LIN {X 0,Y 736.1,Z 322.543,A -85,B 0,C 180,E1 33323.915,E2 33323.915} C_VEL
LIN {X 0,Y 736.031,Z 322.542,A -85,B 0,C 180,E1 33321.184,E2 33321.184} C_VEL
LIN {X 0,Y 736.024,Z 322.538,A -85,B 0,C 180,E1 33318.7,E2 33318.7} C_VEL
LIN {X 0,Y 736.098,Z 322.534,A -85,B 0,C 180,E1 33315.911,E2 33315.911} C_VEL
LIN {X 0,Y 736.039,Z 322.537,A -85,B 0,C 180,E1 33313.033,E2 33313.033} C_VEL
LIN {X 0,Y 736.026,Z 322.539,A -85,B 0,C 180,E1 33310.489,E2 33310.489} C_VEL
LIN {X 0,Y 736.094,Z 322.535,A -85,B 0,C 180,E1 33307.729,E2 33307.729} C_VEL
LIN {X 0,Y 736.045,Z 322.543,A -85,B 0,C 180,E1 33304.831,E2 33304.831} C_VEL
LIN {X 0,Y 736.027,Z 322.536,A -85,B 0,C 180,E1 33302.258,E2 33302.258} C_VEL
LIN {X 0,Y 736.094,Z 322.533,A -85,B 0,C 180,E1 33299.533,E2 33299.533} C_VEL
LIN {X 0,Y 736.044,Z 322.536,A -85,B 0,C 180,E1 33296.573,E2 33296.573} C_VEL
LIN {X 0,Y 736.031,Z 322.539,A -85,B 0,C 180,E1 33293.996,E2 33293.996} C_VEL
LIN {X 0,Y 736.097,Z 322.534,A -85,B 0,C 180,E1 33291.249,E2 33291.249} C_VEL
LIN {X 0,Y 736.097,Z 322.534,A -85,B 0,C 180,E1 33289.048,E2 33289.048} C_VEL
LIN {X 0,Y 735.115,Z 322.666,A -85,B 0,C 180,E1 33288.448,E2 33288.448} C_VEL
LIN {X 0,Y 728.677,Z 323.466,A -85,B 0,C 180,E1 33286.769,E2 33286.769} C_VEL
LIN {X 0,Y 728.112,Z 323.525,A -85,B 0,C 180,E1 33286.333,E2 33286.333} C_VEL
LIN {X 0,Y 728.094,Z 323.528,A -85,B 0,C 180,E1 33283.72,E2 33283.72} C_VEL
LIN {X 0,Y 728.157,Z 323.522,A -85,B 0,C 180,E1 33280.924,E2 33280.924} C_VEL
LIN {X 0,Y 728.106,Z 323.53,A -85,B 0,C 180,E1 33277.981,E2 33277.981} C_VEL
LIN {X 0,Y 728.098,Z 323.526,A -85,B 0,C 180,E1 33275.379,E2 33275.379} C_VEL
LIN {X 0,Y 728.159,Z 323.527,A -85,B 0,C 180,E1 33272.504,E2 33272.504} C_VEL
LIN {X 0,Y 728.102,Z 323.53,A -85,B 0,C 180,E1 33269.644,E2 33269.644} C_VEL
LIN {X 0,Y 728.107,Z 323.529,A -85,B 0,C 180,E1 33267.039,E2 33267.039} C_VEL
LIN {X 0,Y 728.16,Z 323.531,A -85,B 0,C 180,E1 33264.102,E2 33264.102} C_VEL
LIN {X 0,Y 728.107,Z 323.58,A -85,B 0,C 180,E1 33261.311,E2 33261.311} C_VEL
LIN {X 0,Y 729.232,Z 326.748,A -85,B 0,C 180,E1 33260.997,E2 33260.997} C_VEL
LIN {X 0,Y 733.452,Z 336.26,A -85,B 0,C 180,E1 33260.007,E2 33260.007} C_VEL
LIN {X 0,Y 733.535,Z 341.384,A -85,B 0,C 180,E1 33259.674,E2 33259.674} C_VEL
LIN {X 0,Y 735.852,Z 350.383,A -85,B 0,C 180,E1 33259.391,E2 33259.391} C_VEL
LIN {X 0,Y 734.942,Z 560.635,A -85,B 0,C 180,E1 33256.782,E2 33256.782} C_VEL
LIN {X 0,Y 734.06,Z 784.489,A -85,B 0,C 180,E1 33254.097,E2 33254.097} C_VEL
LIN {X 0,Y 733.842,Z 824.081,A -85,B 0,C 180,E1 33253.594,E2 33253.594} C_VEL
LIN {X 0,Y 733.512,Z 850.633,A -85,B 0,C 180,E1 33253.099,E2 33253.099} C_VEL
LIN {X 0,Y 733.193,Z 876.497,A -85,B 0,C 180,E1 33252.467,E2 33252.467} C_VEL
LIN {X 0,Y 732.75,Z 904.112,A -85,B 0,C 180,E1 33251.617,E2 33251.617} C_VEL
LIN {X 0,Y 732.239,Z 928.977,A -85,B 0,C 180,E1 33250.694,E2 33250.694} C_VEL
LIN {X 0,Y 731.795,Z 951.691,A -85,B 0,C 180,E1 33249.712,E2 33249.712} C_VEL
LIN {X 0,Y 731.337,Z 975.92,A -85,B 0,C 180,E1 33248.517,E2 33248.517} C_VEL
LIN {X 0,Y 730.768,Z 999.778,A -85,B 0,C 180,E1 33247.162,E2 33247.162} C_VEL
LIN {X 0,Y 730.337,Z 1020.658,A -85,B 0,C 180,E1 33245.826,E2 33245.826} C_VEL
LIN {X 0,Y 729.892,Z 1043.125,A -85,B 0,C 180,E1 33244.217,E2 33244.217} C_VEL
LIN {X 0,Y 729.439,Z 1063.156,A -85,B 0,C 180,E1 33242.595,E2 33242.595} C_VEL
LIN {X 0,Y 729.121,Z 1082.465,A -85,B 0,C 180,E1 33240.854,E2 33240.854} C_VEL
LIN {X 0,Y 728.788,Z 1100.104,A -85,B 0,C 180,E1 33239.056,E2 33239.056} C_VEL
LIN {X 0,Y 728.566,Z 1114.981,A -85,B 0,C 180,E1 33237.37,E2 33237.37} C_VEL
LIN {X 0,Y 728.345,Z 1130.773,A -85,B 0,C 180,E1 33235.36,E2 33235.36} C_VEL
LIN {X 0,Y 728.172,Z 1143.719,A -85,B 0,C 180,E1 33233.466,E2 33233.466} C_VEL
LIN {X 0,Y 728.099,Z 1154.015,A -85,B 0,C 180,E1 33231.763,E2 33231.763} C_VEL
LIN {X 0,Y 728.021,Z 1163.405,A -85,B 0,C 180,E1 33229.997,E2 33229.997} C_VEL
LIN {X 0,Y 727.956,Z 1173.511,A -85,B 0,C 180,E1 33227.753,E2 33227.753} C_VEL
LIN {X 0,Y 727.938,Z 1181.236,A -85,B 0,C 180,E1 33225.618,E2 33225.618} C_VEL
LIN {X 0,Y 727.921,Z 1187.251,A -85,B 0,C 180,E1 33223.46,E2 33223.46} C_VEL
LIN {X 0,Y 727.912,Z 1191.364,A -85,B 0,C 180,E1 33221.408,E2 33221.408} C_VEL
LIN {X 0,Y 727.912,Z 1193.964,A -85,B 0,C 180,E1 33219.328,E2 33219.328} C_VEL
LIN {X 0,Y 727.912,Z 1194.92,A -85,B 0,C 180,E1 33217.26,E2 33217.26} C_VEL
LIN {X 0,Y 727.914,Z 1194.252,A -85,B 0,C 180,E1 33214.964,E2 33214.964} C_VEL
LIN {X 0,Y 727.911,Z 1192.016,A -85,B 0,C 180,E1 33212.913,E2 33212.913} C_VEL
LIN {X 0,Y 727.916,Z 1187.872,A -85,B 0,C 180,E1 33210.708,E2 33210.708} C_VEL
LIN {X 0,Y 727.926,Z 1182.373,A -85,B 0,C 180,E1 33208.662,E2 33208.662} C_VEL
LIN {X 0,Y 727.944,Z 1175.333,A -85,B 0,C 180,E1 33206.614,E2 33206.614} C_VEL
LIN {X 0,Y 728.001,Z 1165.854,A -85,B 0,C 180,E1 33204.404,E2 33204.404} C_VEL
LIN {X 0,Y 728.074,Z 1155.152,A -85,B 0,C 180,E1 33202.345,E2 33202.345} C_VEL
LIN {X 0,Y 728.186,Z 1144.682,A -85,B 0,C 180,E1 33200.596,E2 33200.596} C_VEL
LIN {X 0,Y 728.307,Z 1133.374,A -85,B 0,C 180,E1 33198.919,E2 33198.919} C_VEL
LIN {X 0,Y 728.51,Z 1118.777,A -85,B 0,C 180,E1 33196.992,E2 33196.992} C_VEL
LIN {X 0,Y 728.753,Z 1102.69,A -85,B 0,C 180,E1 33195.134,E2 33195.134} C_VEL
LIN {X 0,Y 729.006,Z 1086.805,A -85,B 0,C 180,E1 33193.484,E2 33193.484} C_VEL
LIN {X 0,Y 729.398,Z 1067.238,A -85,B 0,C 180,E1 33191.664,E2 33191.664} C_VEL
LIN {X 0,Y 729.751,Z 1047.592,A -85,B 0,C 180,E1 33190.043,E2 33190.043} C_VEL
LIN {X 0,Y 730.245,Z 1026.396,A -85,B 0,C 180,E1 33188.473,E2 33188.473} C_VEL
LIN {X 0,Y 730.684,Z 1003.949,A -85,B 0,C 180,E1 33187.004,E2 33187.004} C_VEL
LIN {X 0,Y 731.156,Z 982.23,A -85,B 0,C 180,E1 33185.737,E2 33185.737} C_VEL
LIN {X 0,Y 731.746,Z 956.143,A -85,B 0,C 180,E1 33184.403,E2 33184.403} C_VEL
LIN {X 0,Y 732.18,Z 932.146,A -85,B 0,C 180,E1 33183.346,E2 33183.346} C_VEL
LIN {X 0,Y 732.629,Z 908.406,A -85,B 0,C 180,E1 33182.442,E2 33182.442} C_VEL
LIN {X 0,Y 733.122,Z 879.506,A -85,B 0,C 180,E1 33181.527,E2 33181.527} C_VEL
LIN {X 0,Y 733.503,Z 853.369,A -85,B 0,C 180,E1 33180.872,E2 33180.872} C_VEL
LIN {X 0,Y 733.788,Z 827.264,A -85,B 0,C 180,E1 33180.368,E2 33180.368} C_VEL
LIN {X 0,Y 734.01,Z 796.894,A -85,B 0,C 180,E1 33179.959,E2 33179.959} C_VEL
LIN {X 0,Y 734.878,Z 575.636,A -85,B 0,C 180,E1 33177.311,E2 33177.311} C_VEL
LIN {X 0,Y 735.783,Z 363.377,A -85,B 0,C 180,E1 33174.683,E2 33174.683} C_VEL
LIN {X 0,Y 735.679,Z 349.285,A -85,B 0,C 180,E1 33174.493,E2 33174.493} C_VEL
LIN {X 0,Y 733.334,Z 340.674,A -85,B 0,C 180,E1 33174.203,E2 33174.203} C_VEL
LIN {X 0,Y 733.221,Z 335.527,A -85,B 0,C 180,E1 33173.834,E2 33173.834} C_VEL
LIN {X 0,Y 728.136,Z 323.997,A -85,B 0,C 180,E1 33172.631,E2 33172.631} C_VEL
LIN {X 0,Y 728.074,Z 323.541,A -85,B 0,C 180,E1 33172.541,E2 33172.541} C_VEL
LIN {X 0,Y 728.091,Z 323.534,A -85,B 0,C 180,E1 33169.492,E2 33169.492} C_VEL
LIN {X 0,Y 728.058,Z 323.536,A -85,B 0,C 180,E1 33167.055,E2 33167.055} C_VEL
LIN {X 0,Y 728.051,Z 323.535,A -85,B 0,C 180,E1 33164.764,E2 33164.764} C_VEL
LIN {X 0,Y 728.064,Z 323.531,A -85,B 0,C 180,E1 33162.401,E2 33162.401} C_VEL
LIN {X 0,Y 728.153,Z 323.531,A -85,B 0,C 180,E1 33159.581,E2 33159.581} C_VEL
LIN {X 0,Y 728.061,Z 323.533,A -85,B 0,C 180,E1 33156.783,E2 33156.783} C_VEL
LIN {X 0,Y 728.055,Z 323.531,A -85,B 0,C 180,E1 33154.46,E2 33154.46} C_VEL
LIN {X 0,Y 728.071,Z 323.533,A -85,B 0,C 180,E1 33152.079,E2 33152.079} C_VEL
LIN {X 0,Y 728.129,Z 323.525,A -85,B 0,C 180,E1 33149.15,E2 33149.15} C_VEL
LIN {X 0,Y 728.063,Z 323.529,A -85,B 0,C 180,E1 33146.509,E2 33146.509} C_VEL
LIN {X 0,Y 728.059,Z 323.533,A -85,B 0,C 180,E1 33144.159,E2 33144.159} C_VEL
LIN {X 0,Y 728.076,Z 323.525,A -85,B 0,C 180,E1 33141.765,E2 33141.765} C_VEL
LIN {X 0,Y 728.123,Z 323.531,A -85,B 0,C 180,E1 33138.827,E2 33138.827} C_VEL
LIN {X 0,Y 728.063,Z 323.531,A -85,B 0,C 180,E1 33136.188,E2 33136.188} C_VEL
LIN {X 0,Y 728.062,Z 323.532,A -85,B 0,C 180,E1 33133.849,E2 33133.849} C_VEL
LIN {X 0,Y 728.097,Z 323.533,A -85,B 0,C 180,E1 33131.325,E2 33131.325} C_VEL
LIN {X 0,Y 728.09,Z 323.531,A -85,B 0,C 180,E1 33128.291,E2 33128.291} C_VEL
LIN {X 0,Y 728.063,Z 323.53,A -85,B 0,C 180,E1 33125.833,E2 33125.833} C_VEL
LIN {X 0,Y 728.065,Z 323.532,A -85,B 0,C 180,E1 33123.543,E2 33123.543} C_VEL
LIN {X 0,Y 728.129,Z 323.533,A -85,B 0,C 180,E1 33120.866,E2 33120.866} C_VEL
LIN {X 0,Y 728.085,Z 323.531,A -85,B 0,C 180,E1 33117.954,E2 33117.954} C_VEL
LIN {X 0,Y 728.065,Z 323.529,A -85,B 0,C 180,E1 33115.51,E2 33115.51} C_VEL
LIN {X 0,Y 728.074,Z 323.532,A -85,B 0,C 180,E1 33113.138,E2 33113.138} C_VEL
LIN {X 0,Y 728.161,Z 323.529,A -85,B 0,C 180,E1 33110.276,E2 33110.276} C_VEL
LIN {X 0,Y 728.072,Z 323.521,A -85,B 0,C 180,E1 33107.468,E2 33107.468} C_VEL
LIN {X 0,Y 728.068,Z 323.53,A -85,B 0,C 180,E1 33105.119,E2 33105.119} C_VEL
LIN {X 0,Y 728.104,Z 323.533,A -85,B 0,C 180,E1 33102.58,E2 33102.58} C_VEL
LIN {X 0,Y 728.092,Z 323.528,A -85,B 0,C 180,E1 33099.481,E2 33099.481} C_VEL
LIN {X 0,Y 728.071,Z 323.53,A -85,B 0,C 180,E1 33097.044,E2 33097.044} C_VEL
LIN {X 0,Y 728.08,Z 323.523,A -85,B 0,C 180,E1 33094.629,E2 33094.629} C_VEL
LIN {X 0,Y 728.159,Z 323.528,A -85,B 0,C 180,E1 33091.722,E2 33091.722} C_VEL
LIN {X 0,Y 728.078,Z 323.529,A -85,B 0,C 180,E1 33088.973,E2 33088.973} C_VEL
LIN {X 0,Y 728.074,Z 323.53,A -85,B 0,C 180,E1 33086.584,E2 33086.584} C_VEL
LIN {X 0,Y 728.143,Z 323.534,A -85,B 0,C 180,E1 33083.844,E2 33083.844} C_VEL
LIN {X 0,Y 728.088,Z 323.533,A -85,B 0,C 180,E1 33080.886,E2 33080.886} C_VEL
LIN {X 0,Y 728.075,Z 323.533,A -85,B 0,C 180,E1 33078.446,E2 33078.446} C_VEL
LIN {X 0,Y 728.11,Z 323.537,A -85,B 0,C 180,E1 33075.873,E2 33075.873} C_VEL
LIN {X 0,Y 728.146,Z 323.695,A -85,B 0,C 180,E1 33075.022,E2 33075.022} C_VEL
LIN {X 0,Y 729.556,Z 327.256,A -85,B 0,C 180,E1 33074.658,E2 33074.658} C_VEL
LIN {X 0,Y 733.673,Z 336.372,A -85,B 0,C 180,E1 33073.705,E2 33073.705} C_VEL
LIN {X 0,Y 733.608,Z 351.232,A -85,B 0,C 180,E1 33072.715,E2 33072.715} C_VEL
LIN {X 0,Y 735.832,Z 360.145,A -85,B 0,C 180,E1 33072.44,E2 33072.44} C_VEL
LIN {X 0,Y 734.944,Z 570.728,A -85,B 0,C 180,E1 33069.826,E2 33069.826} C_VEL
LIN {X 0,Y 734.057,Z 795.931,A -85,B 0,C 180,E1 33067.125,E2 33067.125} C_VEL
LIN {X 0,Y 733.837,Z 834.072,A -85,B 0,C 180,E1 33066.639,E2 33066.639} C_VEL
LIN {X 0,Y 733.515,Z 861.139,A -85,B 0,C 180,E1 33066.133,E2 33066.133} C_VEL
LIN {X 0,Y 733.174,Z 886.975,A -85,B 0,C 180,E1 33065.498,E2 33065.498} C_VEL
LIN {X 0,Y 732.729,Z 915.127,A -85,B 0,C 180,E1 33064.627,E2 33064.627} C_VEL
LIN {X 0,Y 732.218,Z 939.494,A -85,B 0,C 180,E1 33063.716,E2 33063.716} C_VEL
LIN {X 0,Y 731.8,Z 960.602,A -85,B 0,C 180,E1 33062.807,E2 33062.807} C_VEL
LIN {X 0,Y 731.386,Z 982.099,A -85,B 0,C 180,E1 33061.757,E2 33061.757} C_VEL
LIN {X 0,Y 730.852,Z 1007.164,A -85,B 0,C 180,E1 33060.365,E2 33060.365} C_VEL
LIN {X 0,Y 730.377,Z 1027.575,A -85,B 0,C 180,E1 33059.077,E2 33059.077} C_VEL
LIN {X 0,Y 729.986,Z 1046.473,A -85,B 0,C 180,E1 33057.755,E2 33057.755} C_VEL
LIN {X 0,Y 729.556,Z 1068.744,A -85,B 0,C 180,E1 33056.012,E2 33056.012} C_VEL
LIN {X 0,Y 729.183,Z 1085.987,A -85,B 0,C 180,E1 33054.5,E2 33054.5} C_VEL
LIN {X 0,Y 728.938,Z 1102.248,A -85,B 0,C 180,E1 33052.927,E2 33052.927} C_VEL
LIN {X 0,Y 728.632,Z 1120.124,A -85,B 0,C 180,E1 33050.987,E2 33050.987} C_VEL
LIN {X 0,Y 728.421,Z 1133.805,A -85,B 0,C 180,E1 33049.318,E2 33049.318} C_VEL
LIN {X 0,Y 728.29,Z 1145.42,A -85,B 0,C 180,E1 33047.745,E2 33047.745} C_VEL
LIN {X 0,Y 728.151,Z 1156.94,A -85,B 0,C 180,E1 33046.005,E2 33046.005} C_VEL
LIN {X 0,Y 728.047,Z 1169.422,A -85,B 0,C 180,E1 33043.825,E2 33043.825} C_VEL
LIN {X 0,Y 727.972,Z 1178.074,A -85,B 0,C 180,E1 33042.05,E2 33042.05} C_VEL
LIN {X 0,Y 727.953,Z 1185.838,A -85,B 0,C 180,E1 33040.206,E2 33040.206} C_VEL
LIN {X 0,Y 727.927,Z 1193.111,A -85,B 0,C 180,E1 33038.054,E2 33038.054} C_VEL
LIN {X 0,Y 727.914,Z 1198.422,A -85,B 0,C 180,E1 33035.992,E2 33035.992} C_VEL
LIN {X 0,Y 727.907,Z 1202.278,A -85,B 0,C 180,E1 33033.859,E2 33033.859} C_VEL
LIN {X 0,Y 727.908,Z 1204.493,A -85,B 0,C 180,E1 33031.653,E2 33031.653} C_VEL
LIN {X 0,Y 727.89,Z 1204.872,A -85,B 0,C 180,E1 33029.528,E2 33029.528} C_VEL
LIN {X 0,Y 727.906,Z 1203.905,A -85,B 0,C 180,E1 33027.559,E2 33027.559} C_VEL
LIN {X 0,Y 727.908,Z 1201.178,A -85,B 0,C 180,E1 33025.43,E2 33025.43} C_VEL
LIN {X 0,Y 727.916,Z 1196.957,A -85,B 0,C 180,E1 33023.374,E2 33023.374} C_VEL
LIN {X 0,Y 727.936,Z 1191.148,A -85,B 0,C 180,E1 33021.31,E2 33021.31} C_VEL
LIN {X 0,Y 727.944,Z 1183.638,A -85,B 0,C 180,E1 33019.234,E2 33019.234} C_VEL
LIN {X 0,Y 728.028,Z 1173.527,A -85,B 0,C 180,E1 33016.983,E2 33016.983} C_VEL
LIN {X 0,Y 728.084,Z 1164.528,A -85,B 0,C 180,E1 33015.282,E2 33015.282} C_VEL
LIN {X 0,Y 728.169,Z 1154.741,A -85,B 0,C 180,E1 33013.651,E2 33013.651} C_VEL
LIN {X 0,Y 728.298,Z 1144.115,A -85,B 0,C 180,E1 33012.07,E2 33012.07} C_VEL
LIN {X 0,Y 728.489,Z 1130.976,A -85,B 0,C 180,E1 33010.318,E2 33010.318} C_VEL
LIN {X 0,Y 728.74,Z 1113.473,A -85,B 0,C 180,E1 33008.265,E2 33008.265} C_VEL
LIN {X 0,Y 728.955,Z 1098.833,A -85,B 0,C 180,E1 33006.732,E2 33006.732} C_VEL
LIN {X 0,Y 729.277,Z 1082.529,A -85,B 0,C 180,E1 33005.183,E2 33005.183} C_VEL
LIN {X 0,Y 729.687,Z 1061.274,A -85,B 0,C 180,E1 33003.38,E2 33003.38} C_VEL
LIN {X 0,Y 730.038,Z 1043.447,A -85,B 0,C 180,E1 33002.025,E2 33002.025} C_VEL
LIN {X 0,Y 730.495,Z 1023.598,A -85,B 0,C 180,E1 33000.659,E2 33000.659} C_VEL
LIN {X 0,Y 731.013,Z 999.732,A -85,B 0,C 180,E1 32999.204,E2 32999.204} C_VEL
LIN {X 0,Y 731.426,Z 978.536,A -85,B 0,C 180,E1 32998.06,E2 32998.06} C_VEL
LIN {X 0,Y 731.862,Z 957.721,A -85,B 0,C 180,E1 32997.061,E2 32997.061} C_VEL
LIN {X 0,Y 732.437,Z 932.735,A -85,B 0,C 180,E1 32996.013,E2 32996.013} C_VEL
LIN {X 0,Y 732.844,Z 907.028,A -85,B 0,C 180,E1 32995.109,E2 32995.109} C_VEL
LIN {X 0,Y 733.216,Z 883.775,A -85,B 0,C 180,E1 32994.416,E2 32994.416} C_VEL
LIN {X 0,Y 733.575,Z 857.308,A -85,B 0,C 180,E1 32993.785,E2 32993.785} C_VEL
LIN {X 0,Y 733.855,Z 829.91,A -85,B 0,C 180,E1 32993.298,E2 32993.298} C_VEL
LIN {X 0,Y 734.293,Z 733.648,A -85,B 0,C 180,E1 32992.137,E2 32992.137} C_VEL
LIN {X 0,Y 735.2,Z 510.796,A -85,B 0,C 180,E1 32989.44,E2 32989.44} C_VEL
LIN {X 0,Y 735.69,Z 358.849,A -85,B 0,C 180,E1 32987.533,E2 32987.533} C_VEL
LIN {X 0,Y 733.48,Z 350.376,A -85,B 0,C 180,E1 32987.246,E2 32987.246} C_VEL
LIN {X 0,Y 733.542,Z 335.96,A -85,B 0,C 180,E1 32986.257,E2 32986.257} C_VEL
LIN {X 0,Y 728.193,Z 324.003,A -85,B 0,C 180,E1 32985.004,E2 32985.004} C_VEL
LIN {X 0,Y 728.129,Z 323.534,A -85,B 0,C 180,E1 32984.944,E2 32984.944} C_VEL
LIN {X 0,Y 728.097,Z 323.536,A -85,B 0,C 180,E1 32981.901,E2 32981.901} C_VEL
LIN {X 0,Y 728.079,Z 323.533,A -85,B 0,C 180,E1 32979.381,E2 32979.381} C_VEL
LIN {X 0,Y 728.119,Z 323.529,A -85,B 0,C 180,E1 32976.78,E2 32976.78} C_VEL
LIN {X 0,Y 728.101,Z 323.533,A -85,B 0,C 180,E1 32973.698,E2 32973.698} C_VEL
LIN {X 0,Y 728.081,Z 323.524,A -85,B 0,C 180,E1 32971.18,E2 32971.18} C_VEL
LIN {X 0,Y 728.109,Z 323.528,A -85,B 0,C 180,E1 32968.638,E2 32968.638} C_VEL
LIN {X 0,Y 728.113,Z 323.533,A -85,B 0,C 180,E1 32965.544,E2 32965.544} C_VEL
LIN {X 0,Y 728.082,Z 323.524,A -85,B 0,C 180,E1 32962.956,E2 32962.956} C_VEL
LIN {X 0,Y 728.12,Z 323.526,A -85,B 0,C 180,E1 32960.33,E2 32960.33} C_VEL
LIN {X 0,Y 728.109,Z 323.528,A -85,B 0,C 180,E1 32957.255,E2 32957.255} C_VEL
LIN {X 0,Y 728.085,Z 323.53,A -85,B 0,C 180,E1 32954.718,E2 32954.718} C_VEL
LIN {X 0,Y 728.117,Z 323.519,A -85,B 0,C 180,E1 32952.117,E2 32952.117} C_VEL
LIN {X 0,Y 728.11,Z 323.531,A -85,B 0,C 180,E1 32949.007,E2 32949.007} C_VEL
LIN {X 0,Y 728.086,Z 323.523,A -85,B 0,C 180,E1 32946.466,E2 32946.466} C_VEL
LIN {X 0,Y 728.133,Z 323.526,A -85,B 0,C 180,E1 32943.779,E2 32943.779} C_VEL
LIN {X 0,Y 728.107,Z 323.528,A -85,B 0,C 180,E1 32940.708,E2 32940.708} C_VEL
LIN {X 0,Y 728.092,Z 323.528,A -85,B 0,C 180,E1 32938.111,E2 32938.111} C_VEL
LIN {X 0,Y 728.158,Z 323.517,A -85,B 0,C 180,E1 32935.353,E2 32935.353} C_VEL
LIN {X 0,Y 728.105,Z 323.529,A -85,B 0,C 180,E1 32932.424,E2 32932.424} C_VEL
LIN {X 0,Y 728.092,Z 323.523,A -85,B 0,C 180,E1 32929.876,E2 32929.876} C_VEL
LIN {X 0,Y 728.159,Z 323.526,A -85,B 0,C 180,E1 32927.066,E2 32927.066} C_VEL
LIN {X 0,Y 728.112,Z 323.525,A -85,B 0,C 180,E1 32926.333,E2 32926.333} C_VEL
LIN {X 0,Y 727.081,Z 323.649,A -85,B 0,C 180,E1 32925.727,E2 32925.727} C_VEL
LIN {X 0,Y 720.669,Z 324.457,A -85,B 0,C 180,E1 32924.028,E2 32924.028} C_VEL
LIN {X 0,Y 720.16,Z 324.516,A -85,B 0,C 180,E1 32923.587,E2 32923.587} C_VEL
LIN {X 0,Y 720.22,Z 324.511,A -85,B 0,C 180,E1 32920.706,E2 32920.706} C_VEL
LIN {X 0,Y 720.162,Z 324.518,A -85,B 0,C 180,E1 32917.897,E2 32917.897} C_VEL
LIN {X 0,Y 720.163,Z 324.514,A -85,B 0,C 180,E1 32915.297,E2 32915.297} C_VEL
LIN {X 0,Y 720.221,Z 324.52,A -85,B 0,C 180,E1 32912.339,E2 32912.339} C_VEL
LIN {X 0,Y 720.161,Z 324.519,A -85,B 0,C 180,E1 32909.55,E2 32909.55} C_VEL
LIN {X 0,Y 720.177,Z 324.518,A -85,B 0,C 180,E1 32906.931,E2 32906.931} C_VEL
LIN {X 0,Y 720.2,Z 324.523,A -85,B 0,C 180,E1 32903.839,E2 32903.839} C_VEL
LIN {X 0,Y 720.231,Z 324.692,A -85,B 0,C 180,E1 32901.845,E2 32901.845} C_VEL
LIN {X 0,Y 721.419,Z 327.919,A -85,B 0,C 180,E1 32901.514,E2 32901.514} C_VEL
LIN {X 0,Y 726.87,Z 339.92,A -85,B 0,C 180,E1 32900.233,E2 32900.233} C_VEL
LIN {X 0,Y 727.128,Z 341.886,A -85,B 0,C 180,E1 32900.135,E2 32900.135} C_VEL
LIN {X 0,Y 729.922,Z 352.615,A -85,B 0,C 180,E1 32899.788,E2 32899.788} C_VEL
LIN {X 0,Y 728.778,Z 562.579,A -85,B 0,C 180,E1 32897.163,E2 32897.163} C_VEL
LIN {X 0,Y 727.665,Z 786.421,A -85,B 0,C 180,E1 32894.456,E2 32894.456} C_VEL
LIN {X 0,Y 727.394,Z 824.658,A -85,B 0,C 180,E1 32893.964,E2 32893.964} C_VEL
LIN {X 0,Y 726.983,Z 851.311,A -85,B 0,C 180,E1 32893.46,E2 32893.46} C_VEL
LIN {X 0,Y 726.578,Z 877.004,A -85,B 0,C 180,E1 32892.825,E2 32892.825} C_VEL
LIN {X 0,Y 726.032,Z 904.199,A -85,B 0,C 180,E1 32891.981,E2 32891.981} C_VEL
LIN {X 0,Y 725.398,Z 929.465,A -85,B 0,C 180,E1 32891.035,E2 32891.035} C_VEL
LIN {X 0,Y 724.81,Z 953.068,A -85,B 0,C 180,E1 32890.003,E2 32890.003} C_VEL
LIN {X 0,Y 724.2,Z 977.808,A -85,B 0,C 180,E1 32888.759,E2 32888.759} C_VEL
LIN {X 0,Y 723.539,Z 1000.552,A -85,B 0,C 180,E1 32887.447,E2 32887.447} C_VEL
LIN {X 0,Y 722.967,Z 1022.137,A -85,B 0,C 180,E1 32886.048,E2 32886.048} C_VEL
LIN {X 0,Y 722.359,Z 1045.479,A -85,B 0,C 180,E1 32884.336,E2 32884.336} C_VEL
LIN {X 0,Y 721.828,Z 1065.309,A -85,B 0,C 180,E1 32882.698,E2 32882.698} C_VEL
LIN {X 0,Y 721.36,Z 1085.563,A -85,B 0,C 180,E1 32880.817,E2 32880.817} C_VEL
LIN {X 0,Y 721,Z 1101.914,A -85,B 0,C 180,E1 32879.109,E2 32879.109} C_VEL
LIN {X 0,Y 720.71,Z 1118.213,A -85,B 0,C 180,E1 32877.214,E2 32877.214} C_VEL
LIN {X 0,Y 720.433,Z 1133.216,A -85,B 0,C 180,E1 32875.218,E2 32875.218} C_VEL
LIN {X 0,Y 720.24,Z 1144.814,A -85,B 0,C 180,E1 32873.479,E2 32873.479} C_VEL
LIN {X 0,Y 720.144,Z 1155.107,A -85,B 0,C 180,E1 32871.738,E2 32871.738} C_VEL
LIN {X 0,Y 720.048,Z 1165.905,A -85,B 0,C 180,E1 32869.636,E2 32869.636} C_VEL
LIN {X 0,Y 719.963,Z 1175.478,A -85,B 0,C 180,E1 32867.373,E2 32867.373} C_VEL
LIN {X 0,Y 719.932,Z 1182.494,A -85,B 0,C 180,E1 32865.3,E2 32865.3} C_VEL
LIN {X 0,Y 719.92,Z 1187.923,A -85,B 0,C 180,E1 32863.248,E2 32863.248} C_VEL
LIN {X 0,Y 719.911,Z 1192.003,A -85,B 0,C 180,E1 32861.05,E2 32861.05} C_VEL
LIN {X 0,Y 719.911,Z 1194.265,A -85,B 0,C 180,E1 32858.949,E2 32858.949} C_VEL
LIN {X 0,Y 719.903,Z 1194.913,A -85,B 0,C 180,E1 32856.62,E2 32856.62} C_VEL
LIN {X 0,Y 719.906,Z 1193.949,A -85,B 0,C 180,E1 32854.541,E2 32854.541} C_VEL
LIN {X 0,Y 719.912,Z 1191.264,A -85,B 0,C 180,E1 32852.388,E2 32852.388} C_VEL
LIN {X 0,Y 719.923,Z 1187.106,A -85,B 0,C 180,E1 32850.318,E2 32850.318} C_VEL
LIN {X 0,Y 719.945,Z 1181.154,A -85,B 0,C 180,E1 32848.17,E2 32848.17} C_VEL
LIN {X 0,Y 719.982,Z 1173.131,A -85,B 0,C 180,E1 32845.939,E2 32845.939} C_VEL
LIN {X 0,Y 720.065,Z 1163.489,A -85,B 0,C 180,E1 32843.782,E2 32843.782} C_VEL
LIN {X 0,Y 720.128,Z 1154.245,A -85,B 0,C 180,E1 32842.019,E2 32842.019} C_VEL
LIN {X 0,Y 720.262,Z 1143.873,A -85,B 0,C 180,E1 32840.282,E2 32840.282} C_VEL
LIN {X 0,Y 720.481,Z 1131.121,A -85,B 0,C 180,E1 32838.391,E2 32838.391} C_VEL
LIN {X 0,Y 720.739,Z 1115.415,A -85,B 0,C 180,E1 32836.359,E2 32836.359} C_VEL
LIN {X 0,Y 721.012,Z 1100.457,A -85,B 0,C 180,E1 32834.641,E2 32834.641} C_VEL
LIN {X 0,Y 721.433,Z 1083.767,A -85,B 0,C 180,E1 32832.913,E2 32832.913} C_VEL
LIN {X 0,Y 721.853,Z 1063.872,A -85,B 0,C 180,E1 32831.088,E2 32831.088} C_VEL
LIN {X 0,Y 722.4,Z 1044.042,A -85,B 0,C 180,E1 32829.46,E2 32829.46} C_VEL
LIN {X 0,Y 722.976,Z 1021.489,A -85,B 0,C 180,E1 32827.818,E2 32827.818} C_VEL
LIN {X 0,Y 723.573,Z 999.846,A -85,B 0,C 180,E1 32826.419,E2 32826.419} C_VEL
LIN {X 0,Y 724.267,Z 975.235,A -85,B 0,C 180,E1 32825.012,E2 32825.012} C_VEL
LIN {X 0,Y 724.847,Z 950.914,A -85,B 0,C 180,E1 32823.806,E2 32823.806} C_VEL
LIN {X 0,Y 725.456,Z 927.951,A -85,B 0,C 180,E1 32822.814,E2 32822.814} C_VEL
LIN {X 0,Y 726.104,Z 901.508,A -85,B 0,C 180,E1 32821.838,E2 32821.838} C_VEL
LIN {X 0,Y 726.608,Z 874.713,A -85,B 0,C 180,E1 32821.023,E2 32821.023} C_VEL
LIN {X 0,Y 727.031,Z 848.988,A -85,B 0,C 180,E1 32820.401,E2 32820.401} C_VEL
LIN {X 0,Y 727.405,Z 822.47,A -85,B 0,C 180,E1 32819.912,E2 32819.912} C_VEL
LIN {X 0,Y 727.721,Z 774.785,A -85,B 0,C 180,E1 32819.315,E2 32819.315} C_VEL
LIN {X 0,Y 728.848,Z 550.056,A -85,B 0,C 180,E1 32816.594,E2 32816.594} C_VEL
LIN {X 0,Y 729.892,Z 351.989,A -85,B 0,C 180,E1 32814.111,E2 32814.111} C_VEL
LIN {X 0,Y 726.812,Z 340.648,A -85,B 0,C 180,E1 32813.724,E2 32813.724} C_VEL
LIN {X 0,Y 726.364,Z 338.985,A -85,B 0,C 180,E1 32813.573,E2 32813.573} C_VEL
LIN {X 0,Y 720.269,Z 324.967,A -85,B 0,C 180,E1 32812.088,E2 32812.088} C_VEL
LIN {X 0,Y 720.209,Z 324.522,A -85,B 0,C 180,E1 32812.047,E2 32812.047} C_VEL
LIN {X 0,Y 720.122,Z 324.524,A -85,B 0,C 180,E1 32809.177,E2 32809.177} C_VEL
LIN {X 0,Y 720.115,Z 324.526,A -85,B 0,C 180,E1 32806.8,E2 32806.8} C_VEL
LIN {X 0,Y 720.128,Z 324.525,A -85,B 0,C 180,E1 32804.411,E2 32804.411} C_VEL
LIN {X 0,Y 720.185,Z 324.521,A -85,B 0,C 180,E1 32801.473,E2 32801.473} C_VEL
LIN {X 0,Y 720.121,Z 324.523,A -85,B 0,C 180,E1 32798.838,E2 32798.838} C_VEL
LIN {X 0,Y 720.117,Z 324.522,A -85,B 0,C 180,E1 32796.494,E2 32796.494} C_VEL
LIN {X 0,Y 720.143,Z 324.521,A -85,B 0,C 180,E1 32794.016,E2 32794.016} C_VEL
LIN {X 0,Y 720.145,Z 324.522,A -85,B 0,C 180,E1 32790.903,E2 32790.903} C_VEL
LIN {X 0,Y 720.119,Z 324.513,A -85,B 0,C 180,E1 32788.441,E2 32788.441} C_VEL
LIN {X 0,Y 720.126,Z 324.519,A -85,B 0,C 180,E1 32786.061,E2 32786.061} C_VEL
LIN {X 0,Y 720.219,Z 324.513,A -85,B 0,C 180,E1 32783.215,E2 32783.215} C_VEL
LIN {X 0,Y 720.128,Z 324.517,A -85,B 0,C 180,E1 32780.396,E2 32780.396} C_VEL
LIN {X 0,Y 720.121,Z 324.522,A -85,B 0,C 180,E1 32778.037,E2 32778.037} C_VEL
LIN {X 0,Y 720.137,Z 324.521,A -85,B 0,C 180,E1 32775.626,E2 32775.626} C_VEL
LIN {X 0,Y 720.187,Z 324.52,A -85,B 0,C 180,E1 32772.672,E2 32772.672} C_VEL
LIN {X 0,Y 720.126,Z 324.518,A -85,B 0,C 180,E1 32769.995,E2 32769.995} C_VEL
LIN {X 0,Y 720.127,Z 324.521,A -85,B 0,C 180,E1 32767.66,E2 32767.66} C_VEL
LIN {X 0,Y 720.168,Z 324.52,A -85,B 0,C 180,E1 32765.098,E2 32765.098} C_VEL
LIN {X 0,Y 720.147,Z 324.519,A -85,B 0,C 180,E1 32762.069,E2 32762.069} C_VEL
LIN {X 0,Y 720.126,Z 324.519,A -85,B 0,C 180,E1 32759.602,E2 32759.602} C_VEL
LIN {X 0,Y 720.137,Z 324.522,A -85,B 0,C 180,E1 32757.215,E2 32757.215} C_VEL
LIN {X 0,Y 720.217,Z 324.519,A -85,B 0,C 180,E1 32754.343,E2 32754.343} C_VEL
LIN {X 0,Y 720.132,Z 324.519,A -85,B 0,C 180,E1 32751.536,E2 32751.536} C_VEL
LIN {X 0,Y 720.129,Z 324.52,A -85,B 0,C 180,E1 32749.196,E2 32749.196} C_VEL
LIN {X 0,Y 720.175,Z 324.509,A -85,B 0,C 180,E1 32746.593,E2 32746.593} C_VEL
LIN {X 0,Y 720.156,Z 324.519,A -85,B 0,C 180,E1 32743.612,E2 32743.612} C_VEL
LIN {X 0,Y 720.13,Z 324.51,A -85,B 0,C 180,E1 32741.124,E2 32741.124} C_VEL
LIN {X 0,Y 720.144,Z 324.52,A -85,B 0,C 180,E1 32738.689,E2 32738.689} C_VEL
LIN {X 0,Y 720.212,Z 324.505,A -85,B 0,C 180,E1 32735.797,E2 32735.797} C_VEL
LIN {X 0,Y 720.137,Z 324.52,A -85,B 0,C 180,E1 32733.046,E2 32733.046} C_VEL
LIN {X 0,Y 720.137,Z 324.52,A -85,B 0,C 180,E1 32730.651,E2 32730.651} C_VEL
LIN {X 0,Y 720.214,Z 324.523,A -85,B 0,C 180,E1 32727.87,E2 32727.87} C_VEL
LIN {X 0,Y 720.149,Z 324.52,A -85,B 0,C 180,E1 32725,E2 32725} C_VEL
LIN {X 0,Y 720.136,Z 324.522,A -85,B 0,C 180,E1 32722.544,E2 32722.544} C_VEL
LIN {X 0,Y 720.167,Z 324.527,A -85,B 0,C 180,E1 32719.996,E2 32719.996} C_VEL
LIN {X 0,Y 720.163,Z 324.524,A -85,B 0,C 180,E1 32716.91,E2 32716.91} C_VEL
LIN {X 0,Y 720.213,Z 324.534,A -85,B 0,C 180,E1 32715.595,E2 32715.595} C_VEL
LIN {X 0,Y 721.468,Z 327.926,A -85,B 0,C 180,E1 32715.247,E2 32715.247} C_VEL
LIN {X 0,Y 727.142,Z 340.615,A -85,B 0,C 180,E1 32713.9,E2 32713.9} C_VEL
LIN {X 0,Y 727.071,Z 351.188,A -85,B 0,C 180,E1 32713.193,E2 32713.193} C_VEL
LIN {X 0,Y 729.903,Z 362.188,A -85,B 0,C 180,E1 32712.84,E2 32712.84} C_VEL
LIN {X 0,Y 728.779,Z 572.636,A -85,B 0,C 180,E1 32710.207,E2 32710.207} C_VEL
LIN {X 0,Y 727.664,Z 797.21,A -85,B 0,C 180,E1 32707.492,E2 32707.492} C_VEL
LIN {X 0,Y 727.391,Z 834.662,A -85,B 0,C 180,E1 32707.009,E2 32707.009} C_VEL
LIN {X 0,Y 726.983,Z 862.081,A -85,B 0,C 180,E1 32706.489,E2 32706.489} C_VEL
LIN {X 0,Y 726.55,Z 887.85,A -85,B 0,C 180,E1 32705.846,E2 32705.846} C_VEL
LIN {X 0,Y 725.973,Z 916.212,A -85,B 0,C 180,E1 32704.955,E2 32704.955} C_VEL
LIN {X 0,Y 725.376,Z 939.909,A -85,B 0,C 180,E1 32704.06,E2 32704.06} C_VEL
LIN {X 0,Y 724.836,Z 961.082,A -85,B 0,C 180,E1 32703.139,E2 32703.139} C_VEL
LIN {X 0,Y 724.298,Z 983.241,A -85,B 0,C 180,E1 32702.045,E2 32702.045} C_VEL
LIN {X 0,Y 723.606,Z 1008.626,A -85,B 0,C 180,E1 32700.609,E2 32700.609} C_VEL
LIN {X 0,Y 723.047,Z 1028.239,A -85,B 0,C 180,E1 32699.355,E2 32699.355} C_VEL
LIN {X 0,Y 722.54,Z 1047.296,A -85,B 0,C 180,E1 32698.005,E2 32698.005} C_VEL
LIN {X 0,Y 721.988,Z 1069.76,A -85,B 0,C 180,E1 32696.217,E2 32696.217} C_VEL
LIN {X 0,Y 721.543,Z 1086.385,A -85,B 0,C 180,E1 32694.739,E2 32694.739} C_VEL
LIN {X 0,Y 721.207,Z 1103.097,A -85,B 0,C 180,E1 32693.1,E2 32693.1} C_VEL
LIN {X 0,Y 720.819,Z 1120.837,A -85,B 0,C 180,E1 32691.14,E2 32691.14} C_VEL
LIN {X 0,Y 720.582,Z 1133.807,A -85,B 0,C 180,E1 32689.536,E2 32689.536} C_VEL
LIN {X 0,Y 720.389,Z 1146.004,A -85,B 0,C 180,E1 32687.863,E2 32687.863} C_VEL
LIN {X 0,Y 720.214,Z 1158.903,A -85,B 0,C 180,E1 32685.872,E2 32685.872} C_VEL
LIN {X 0,Y 720.078,Z 1170.244,A -85,B 0,C 180,E1 32683.817,E2 32683.817} C_VEL
LIN {X 0,Y 719.995,Z 1178.432,A -85,B 0,C 180,E1 32682.104,E2 32682.104} C_VEL
LIN {X 0,Y 719.965,Z 1186.135,A -85,B 0,C 180,E1 32680.239,E2 32680.239} C_VEL
LIN {X 0,Y 719.933,Z 1193.544,A -85,B 0,C 180,E1 32678.001,E2 32678.001} C_VEL
LIN {X 0,Y 719.918,Z 1198.937,A -85,B 0,C 180,E1 32675.819,E2 32675.819} C_VEL
LIN {X 0,Y 719.909,Z 1202.484,A -85,B 0,C 180,E1 32673.743,E2 32673.743} C_VEL
LIN {X 0,Y 719.909,Z 1204.549,A -85,B 0,C 180,E1 32671.592,E2 32671.592} C_VEL
LIN {X 0,Y 719.89,Z 1204.872,A -85,B 0,C 180,E1 32669.523,E2 32669.523} C_VEL
LIN {X 0,Y 719.906,Z 1203.902,A -85,B 0,C 180,E1 32667.532,E2 32667.532} C_VEL
LIN {X 0,Y 719.908,Z 1201.178,A -85,B 0,C 180,E1 32665.38,E2 32665.38} C_VEL
LIN {X 0,Y 719.917,Z 1196.832,A -85,B 0,C 180,E1 32663.249,E2 32663.249} C_VEL
LIN {X 0,Y 719.937,Z 1190.891,A -85,B 0,C 180,E1 32661.132,E2 32661.132} C_VEL
LIN {X 0,Y 719.972,Z 1183.001,A -85,B 0,C 180,E1 32658.951,E2 32658.951} C_VEL
LIN {X 0,Y 720.061,Z 1173.152,A -85,B 0,C 180,E1 32656.762,E2 32656.762} C_VEL
LIN {X 0,Y 720.128,Z 1164.064,A -85,B 0,C 180,E1 32655.034,E2 32655.034} C_VEL
LIN {X 0,Y 720.263,Z 1154.221,A -85,B 0,C 180,E1 32653.383,E2 32653.383} C_VEL
LIN {X 0,Y 720.441,Z 1142.511,A -85,B 0,C 180,E1 32651.637,E2 32651.637} C_VEL
LIN {X 0,Y 720.722,Z 1126.521,A -85,B 0,C 180,E1 32649.537,E2 32649.537} C_VEL
LIN {X 0,Y 720.991,Z 1111.843,A -85,B 0,C 180,E1 32647.839,E2 32647.839} C_VEL
LIN {X 0,Y 721.307,Z 1097.128,A -85,B 0,C 180,E1 32646.297,E2 32646.297} C_VEL
LIN {X 0,Y 721.785,Z 1077.881,A -85,B 0,C 180,E1 32644.481,E2 32644.481} C_VEL
LIN {X 0,Y 722.23,Z 1059.06,A -85,B 0,C 180,E1 32642.905,E2 32642.905} C_VEL
LIN {X 0,Y 722.736,Z 1041.03,A -85,B 0,C 180,E1 32641.537,E2 32641.537} C_VEL
LIN {X 0,Y 723.365,Z 1018.082,A -85,B 0,C 180,E1 32639.976,E2 32639.976} C_VEL
LIN {X 0,Y 723.901,Z 996.241,A -85,B 0,C 180,E1 32638.666,E2 32638.666} C_VEL
LIN {X 0,Y 724.472,Z 975.869,A -85,B 0,C 180,E1 32637.576,E2 32637.576} C_VEL
LIN {X 0,Y 725.163,Z 951.713,A -85,B 0,C 180,E1 32636.434,E2 32636.434} C_VEL
LIN {X 0,Y 725.714,Z 926.414,A -85,B 0,C 180,E1 32635.415,E2 32635.415} C_VEL
LIN {X 0,Y 726.174,Z 904.863,A -85,B 0,C 180,E1 32634.67,E2 32634.67} C_VEL
LIN {X 0,Y 726.646,Z 881.764,A -85,B 0,C 180,E1 32633.988,E2 32633.988} C_VEL
LIN {X 0,Y 727.127,Z 854.692,A -85,B 0,C 180,E1 32633.354,E2 32633.354} C_VEL
LIN {X 0,Y 727.448,Z 827.377,A -85,B 0,C 180,E1 32632.882,E2 32632.882} C_VEL
LIN {X 0,Y 728.656,Z 595.56,A -85,B 0,C 180,E1 32630.074,E2 32630.074} C_VEL
LIN {X 0,Y 729.735,Z 390.43,A -85,B 0,C 180,E1 32627.518,E2 32627.518} C_VEL
LIN {X 0,Y 729.733,Z 360.849,A -85,B 0,C 180,E1 32627.13,E2 32627.13} C_VEL
LIN {X 0,Y 726.958,Z 350.376,A -85,B 0,C 180,E1 32626.769,E2 32626.769} C_VEL
LIN {X 0,Y 727.031,Z 340.058,A -85,B 0,C 180,E1 32626.053,E2 32626.053} C_VEL
LIN {X 0,Y 721.468,Z 327.926,A -85,B 0,C 180,E1 32624.753,E2 32624.753} C_VEL
LIN {X 0,Y 720.211,Z 324.522,A -85,B 0,C 180,E1 32624.378,E2 32624.378} C_VEL
LIN {X 0,Y 720.145,Z 324.524,A -85,B 0,C 180,E1 32621.672,E2 32621.672} C_VEL
LIN {X 0,Y 720.148,Z 324.522,A -85,B 0,C 180,E1 32619.179,E2 32619.179} C_VEL
LIN {X 0,Y 720.222,Z 324.521,A -85,B 0,C 180,E1 32616.357,E2 32616.357} C_VEL
LIN {X 0,Y 720.151,Z 324.521,A -85,B 0,C 180,E1 32613.546,E2 32613.546} C_VEL
LIN {X 0,Y 720.145,Z 324.511,A -85,B 0,C 180,E1 32611.058,E2 32611.058} C_VEL
LIN {X 0,Y 720.221,Z 324.516,A -85,B 0,C 180,E1 32608.256,E2 32608.256} C_VEL
LIN {X 0,Y 720.154,Z 324.521,A -85,B 0,C 180,E1 32605.318,E2 32605.318} C_VEL
LIN {X 0,Y 720.147,Z 324.511,A -85,B 0,C 180,E1 32602.792,E2 32602.792} C_VEL
LIN {X 0,Y 720.223,Z 324.515,A -85,B 0,C 180,E1 32599.97,E2 32599.97} C_VEL
LIN {X 0,Y 720.152,Z 324.515,A -85,B 0,C 180,E1 32597.035,E2 32597.035} C_VEL
LIN {X 0,Y 720.153,Z 324.518,A -85,B 0,C 180,E1 32594.473,E2 32594.473} C_VEL
LIN {X 0,Y 720.222,Z 324.508,A -85,B 0,C 180,E1 32591.613,E2 32591.613} C_VEL
LIN {X 0,Y 720.155,Z 324.518,A -85,B 0,C 180,E1 32588.785,E2 32588.785} C_VEL
LIN {X 0,Y 720.155,Z 324.509,A -85,B 0,C 180,E1 32586.217,E2 32586.217} C_VEL
LIN {X 0,Y 720.222,Z 324.519,A -85,B 0,C 180,E1 32583.343,E2 32583.343} C_VEL
LIN {X 0,Y 720.153,Z 324.516,A -85,B 0,C 180,E1 32580.477,E2 32580.477} C_VEL
LIN {X 0,Y 720.162,Z 324.516,A -85,B 0,C 180,E1 32577.931,E2 32577.931} C_VEL
LIN {X 0,Y 720.218,Z 324.51,A -85,B 0,C 180,E1 32574.982,E2 32574.982} C_VEL
LIN {X 0,Y 720.153,Z 324.517,A -85,B 0,C 180,E1 32572.18,E2 32572.18} C_VEL
LIN {X 0,Y 720.178,Z 324.509,A -85,B 0,C 180,E1 32569.521,E2 32569.521} C_VEL
LIN {X 0,Y 720.178,Z 324.513,A -85,B 0,C 180,E1 32566.371,E2 32566.371} C_VEL
LIN {X 0,Y 720.156,Z 324.517,A -85,B 0,C 180,E1 32563.712,E2 32563.712} C_VEL
LIN {X 0,Y 720.16,Z 324.516,A -85,B 0,C 180,E1 32563.587,E2 32563.587} C_VEL
LIN {X 0,Y 719.201,Z 324.642,A -85,B 0,C 180,E1 32562.974,E2 32562.974} C_VEL
LIN {X 0,Y 712.809,Z 325.434,A -85,B 0,C 180,E1 32561.258,E2 32561.258} C_VEL
LIN {X 0,Y 712.281,Z 325.498,A -85,B 0,C 180,E1 32560.812,E2 32560.812} C_VEL
LIN {X 0,Y 712.223,Z 325.507,A -85,B 0,C 180,E1 32557.899,E2 32557.899} C_VEL
LIN {X 0,Y 712.227,Z 325.503,A -85,B 0,C 180,E1 32555.269,E2 32555.269} C_VEL
LIN {X 0,Y 712.281,Z 325.51,A -85,B 0,C 180,E1 32552.312,E2 32552.312} C_VEL
LIN {X 0,Y 712.222,Z 325.508,A -85,B 0,C 180,E1 32549.538,E2 32549.538} C_VEL
LIN {X 0,Y 712.252,Z 325.507,A -85,B 0,C 180,E1 32546.804,E2 32546.804} C_VEL
LIN {X 0,Y 712.242,Z 325.514,A -85,B 0,C 180,E1 32543.67,E2 32543.67} C_VEL
LIN {X 0,Y 712.294,Z 325.615,A -85,B 0,C 180,E1 32542.415,E2 32542.415} C_VEL
LIN {X 0,Y 713.661,Z 329.098,A -85,B 0,C 180,E1 32542.043,E2 32542.043} C_VEL
LIN {X 0,Y 719.236,Z 341.291,A -85,B 0,C 180,E1 32540.736,E2 32540.736} C_VEL
LIN {X 0,Y 721.687,Z 345.669,A -85,B 0,C 180,E1 32540.491,E2 32540.491} C_VEL
LIN {X 0,Y 724.029,Z 354.724,A -85,B 0,C 180,E1 32540.194,E2 32540.194} C_VEL
LIN {X 0,Y 722.647,Z 564.35,A -85,B 0,C 180,E1 32537.552,E2 32537.552} C_VEL
LIN {X 0,Y 721.303,Z 787.792,A -85,B 0,C 180,E1 32534.828,E2 32534.828} C_VEL
LIN {X 0,Y 720.975,Z 824.989,A -85,B 0,C 180,E1 32534.343,E2 32534.343} C_VEL
LIN {X 0,Y 720.489,Z 851.685,A -85,B 0,C 180,E1 32533.834,E2 32533.834} C_VEL
LIN {X 0,Y 720.001,Z 877.155,A -85,B 0,C 180,E1 32533.2,E2 32533.2} C_VEL
LIN {X 0,Y 719.352,Z 904.073,A -85,B 0,C 180,E1 32532.359,E2 32532.359} C_VEL
LIN {X 0,Y 718.62,Z 929.228,A -85,B 0,C 180,E1 32531.412,E2 32531.412} C_VEL
LIN {X 0,Y 717.874,Z 953.069,A -85,B 0,C 180,E1 32530.365,E2 32530.365} C_VEL
LIN {X 0,Y 717.107,Z 978.603,A -85,B 0,C 180,E1 32529.066,E2 32529.066} C_VEL
LIN {X 0,Y 716.328,Z 1001.325,A -85,B 0,C 180,E1 32527.739,E2 32527.739} C_VEL
LIN {X 0,Y 715.609,Z 1023.654,A -85,B 0,C 180,E1 32526.271,E2 32526.271} C_VEL
LIN {X 0,Y 714.886,Z 1046.055,A -85,B 0,C 180,E1 32524.6,E2 32524.6} C_VEL
LIN {X 0,Y 714.236,Z 1066.378,A -85,B 0,C 180,E1 32522.899,E2 32522.899} C_VEL
LIN {X 0,Y 713.684,Z 1086.097,A -85,B 0,C 180,E1 32521.035,E2 32521.035} C_VEL
LIN {X 0,Y 713.24,Z 1102.565,A -85,B 0,C 180,E1 32519.291,E2 32519.291} C_VEL
LIN {X 0,Y 712.865,Z 1119.365,A -85,B 0,C 180,E1 32517.3,E2 32517.3} C_VEL
LIN {X 0,Y 712.54,Z 1133.827,A -85,B 0,C 180,E1 32515.34,E2 32515.34} C_VEL
LIN {X 0,Y 712.316,Z 1145.486,A -85,B 0,C 180,E1 32513.561,E2 32513.561} C_VEL
LIN {X 0,Y 712.172,Z 1156.92,A -85,B 0,C 180,E1 32511.582,E2 32511.582} C_VEL
LIN {X 0,Y 712.042,Z 1167.394,A -85,B 0,C 180,E1 32509.439,E2 32509.439} C_VEL
LIN {X 0,Y 711.975,Z 1175.784,A -85,B 0,C 180,E1 32507.405,E2 32507.405} C_VEL
LIN {X 0,Y 711.937,Z 1182.749,A -85,B 0,C 180,E1 32505.309,E2 32505.309} C_VEL
LIN {X 0,Y 711.921,Z 1188.104,A -85,B 0,C 180,E1 32503.234,E2 32503.234} C_VEL
LIN {X 0,Y 711.91,Z 1192.119,A -85,B 0,C 180,E1 32501.012,E2 32501.012} C_VEL
LIN {X 0,Y 711.908,Z 1194.324,A -85,B 0,C 180,E1 32498.887,E2 32498.887} C_VEL
LIN {X 0,Y 711.903,Z 1194.89,A -85,B 0,C 180,E1 32496.532,E2 32496.532} C_VEL
LIN {X 0,Y 711.906,Z 1193.945,A -85,B 0,C 180,E1 32494.511,E2 32494.511} C_VEL
LIN {X 0,Y 711.913,Z 1191.261,A -85,B 0,C 180,E1 32492.334,E2 32492.334} C_VEL
LIN {X 0,Y 711.925,Z 1187.1,A -85,B 0,C 180,E1 32490.241,E2 32490.241} C_VEL
LIN {X 0,Y 711.953,Z 1181.146,A -85,B 0,C 180,E1 32488.068,E2 32488.068} C_VEL
LIN {X 0,Y 712.01,Z 1173.126,A -85,B 0,C 180,E1 32485.812,E2 32485.812} C_VEL
LIN {X 0,Y 712.093,Z 1163.489,A -85,B 0,C 180,E1 32483.631,E2 32483.631} C_VEL
LIN {X 0,Y 712.193,Z 1154.023,A -85,B 0,C 180,E1 32481.808,E2 32481.808} C_VEL
LIN {X 0,Y 712.381,Z 1143.164,A -85,B 0,C 180,E1 32479.977,E2 32479.977} C_VEL
LIN {X 0,Y 712.628,Z 1129.376,A -85,B 0,C 180,E1 32477.933,E2 32477.933} C_VEL
LIN {X 0,Y 712.948,Z 1114.057,A -85,B 0,C 180,E1 32475.959,E2 32475.959} C_VEL
LIN {X 0,Y 713.334,Z 1098.97,A -85,B 0,C 180,E1 32474.221,E2 32474.221} C_VEL
LIN {X 0,Y 713.834,Z 1079.991,A -85,B 0,C 180,E1 32472.27,E2 32472.27} C_VEL
LIN {X 0,Y 714.443,Z 1060.498,A -85,B 0,C 180,E1 32470.502,E2 32470.502} C_VEL
LIN {X 0,Y 715.095,Z 1039.146,A -85,B 0,C 180,E1 32468.769,E2 32468.769} C_VEL
LIN {X 0,Y 715.814,Z 1017.354,A -85,B 0,C 180,E1 32467.21,E2 32467.21} C_VEL
LIN {X 0,Y 716.574,Z 994.975,A -85,B 0,C 180,E1 32465.781,E2 32465.781} C_VEL
LIN {X 0,Y 717.307,Z 971.005,A -85,B 0,C 180,E1 32464.438,E2 32464.438} C_VEL
LIN {X 0,Y 718.051,Z 948.117,A -85,B 0,C 180,E1 32463.316,E2 32463.316} C_VEL
LIN {X 0,Y 718.818,Z 923.611,A -85,B 0,C 180,E1 32462.272,E2 32462.272} C_VEL
LIN {X 0,Y 719.485,Z 897.396,A -85,B 0,C 180,E1 32461.329,E2 32461.329} C_VEL
LIN {X 0,Y 720.061,Z 873.085,A -85,B 0,C 180,E1 32460.6,E2 32460.6} C_VEL
LIN {X 0,Y 720.596,Z 847.254,A -85,B 0,C 180,E1 32459.981,E2 32459.981} C_VEL
LIN {X 0,Y 721.028,Z 819.617,A -85,B 0,C 180,E1 32459.484,E2 32459.484} C_VEL
LIN {X 0,Y 722.458,Z 594.703,A -85,B 0,C 180,E1 32456.733,E2 32456.733} C_VEL
LIN {X 0,Y 723.82,Z 381.695,A -85,B 0,C 180,E1 32454.059,E2 32454.059} C_VEL
LIN {X 0,Y 723.864,Z 353.768,A -85,B 0,C 180,E1 32453.691,E2 32453.691} C_VEL
LIN {X 0,Y 721.081,Z 344.357,A -85,B 0,C 180,E1 32453.356,E2 32453.356} C_VEL
LIN {X 0,Y 718.764,Z 340.686,A -85,B 0,C 180,E1 32453.121,E2 32453.121} C_VEL
LIN {X 0,Y 713.433,Z 328.796,A -85,B 0,C 180,E1 32451.826,E2 32451.826} C_VEL
LIN {X 0,Y 712.204,Z 325.517,A -85,B 0,C 180,E1 32451.466,E2 32451.466} C_VEL
LIN {X 0,Y 712.176,Z 325.513,A -85,B 0,C 180,E1 32449.032,E2 32449.032} C_VEL
LIN {X 0,Y 712.176,Z 325.516,A -85,B 0,C 180,E1 32446.755,E2 32446.755} C_VEL
LIN {X 0,Y 712.206,Z 325.515,A -85,B 0,C 180,E1 32444.248,E2 32444.248} C_VEL
LIN {X 0,Y 712.204,Z 325.512,A -85,B 0,C 180,E1 32441.182,E2 32441.182} C_VEL
LIN {X 0,Y 712.177,Z 325.512,A -85,B 0,C 180,E1 32438.685,E2 32438.685} C_VEL
LIN {X 0,Y 712.185,Z 325.512,A -85,B 0,C 180,E1 32436.307,E2 32436.307} C_VEL
LIN {X 0,Y 712.278,Z 325.511,A -85,B 0,C 180,E1 32433.483,E2 32433.483} C_VEL
LIN {X 0,Y 712.185,Z 325.511,A -85,B 0,C 180,E1 32430.615,E2 32430.615} C_VEL
LIN {X 0,Y 712.179,Z 325.501,A -85,B 0,C 180,E1 32428.325,E2 32428.325} C_VEL
LIN {X 0,Y 712.2,Z 325.508,A -85,B 0,C 180,E1 32425.855,E2 32425.855} C_VEL
LIN {X 0,Y 712.223,Z 325.499,A -85,B 0,C 180,E1 32422.798,E2 32422.798} C_VEL
LIN {X 0,Y 712.184,Z 325.505,A -85,B 0,C 180,E1 32420.291,E2 32420.291} C_VEL
LIN {X 0,Y 712.186,Z 325.511,A -85,B 0,C 180,E1 32417.907,E2 32417.907} C_VEL
LIN {X 0,Y 712.252,Z 325.51,A -85,B 0,C 180,E1 32415.22,E2 32415.22} C_VEL
LIN {X 0,Y 712.196,Z 325.51,A -85,B 0,C 180,E1 32412.239,E2 32412.239} C_VEL
LIN {X 0,Y 712.184,Z 325.507,A -85,B 0,C 180,E1 32409.863,E2 32409.863} C_VEL
LIN {X 0,Y 712.196,Z 325.511,A -85,B 0,C 180,E1 32407.502,E2 32407.502} C_VEL
LIN {X 0,Y 712.273,Z 325.508,A -85,B 0,C 180,E1 32404.59,E2 32404.59} C_VEL
LIN {X 0,Y 712.192,Z 325.509,A -85,B 0,C 180,E1 32401.85,E2 32401.85} C_VEL
LIN {X 0,Y 712.187,Z 325.508,A -85,B 0,C 180,E1 32399.517,E2 32399.517} C_VEL
LIN {X 0,Y 712.224,Z 325.511,A -85,B 0,C 180,E1 32396.942,E2 32396.942} C_VEL
LIN {X 0,Y 712.212,Z 325.509,A -85,B 0,C 180,E1 32393.875,E2 32393.875} C_VEL
LIN {X 0,Y 712.19,Z 325.508,A -85,B 0,C 180,E1 32391.441,E2 32391.441} C_VEL
LIN {X 0,Y 712.195,Z 325.509,A -85,B 0,C 180,E1 32389.074,E2 32389.074} C_VEL
LIN {X 0,Y 712.283,Z 325.497,A -85,B 0,C 180,E1 32386.193,E2 32386.193} C_VEL
LIN {X 0,Y 712.197,Z 325.509,A -85,B 0,C 180,E1 32383.357,E2 32383.357} C_VEL
LIN {X 0,Y 712.195,Z 325.498,A -85,B 0,C 180,E1 32380.906,E2 32380.906} C_VEL
LIN {X 0,Y 712.281,Z 325.51,A -85,B 0,C 180,E1 32378.074,E2 32378.074} C_VEL
LIN {X 0,Y 712.2,Z 325.495,A -85,B 0,C 180,E1 32375.179,E2 32375.179} C_VEL
LIN {X 0,Y 712.199,Z 325.51,A -85,B 0,C 180,E1 32372.706,E2 32372.706} C_VEL
LIN {X 0,Y 712.28,Z 325.51,A -85,B 0,C 180,E1 32369.924,E2 32369.924} C_VEL
LIN {X 0,Y 712.206,Z 325.506,A -85,B 0,C 180,E1 32366.994,E2 32366.994} C_VEL
LIN {X 0,Y 712.199,Z 325.511,A -85,B 0,C 180,E1 32364.514,E2 32364.514} C_VEL
LIN {X 0,Y 712.277,Z 325.512,A -85,B 0,C 180,E1 32361.692,E2 32361.692} C_VEL
LIN {X 0,Y 712.21,Z 325.511,A -85,B 0,C 180,E1 32358.805,E2 32358.805} C_VEL
LIN {X 0,Y 712.201,Z 325.517,A -85,B 0,C 180,E1 32356.303,E2 32356.303} C_VEL
LIN {X 0,Y 712.218,Z 325.607,A -85,B 0,C 180,E1 32356.176,E2 32356.176} C_VEL
LIN {X 0,Y 713.384,Z 328.756,A -85,B 0,C 180,E1 32355.845,E2 32355.845} C_VEL
LIN {X 0,Y 716.061,Z 334.377,A -85,B 0,C 180,E1 32355.213,E2 32355.213} C_VEL
LIN {X 0,Y 720.623,Z 344.746,A -85,B 0,C 180,E1 32354.106,E2 32354.106} C_VEL
LIN {X 0,Y 720.619,Z 351.279,A -85,B 0,C 180,E1 32353.676,E2 32353.676} C_VEL
LIN {X 0,Y 724.01,Z 364.413,A -85,B 0,C 180,E1 32353.245,E2 32353.245} C_VEL
LIN {X 0,Y 722.642,Z 575.258,A -85,B 0,C 180,E1 32350.586,E2 32350.586} C_VEL
LIN {X 0,Y 721.296,Z 799.245,A -85,B 0,C 180,E1 32347.855,E2 32347.855} C_VEL
LIN {X 0,Y 720.973,Z 835.294,A -85,B 0,C 180,E1 32347.384,E2 32347.384} C_VEL
LIN {X 0,Y 720.479,Z 862.712,A -85,B 0,C 180,E1 32346.857,E2 32346.857} C_VEL
LIN {X 0,Y 719.965,Z 888.235,A -85,B 0,C 180,E1 32346.214,E2 32346.214} C_VEL
LIN {X 0,Y 719.265,Z 916.707,A -85,B 0,C 180,E1 32345.311,E2 32345.311} C_VEL
LIN {X 0,Y 718.598,Z 939.502,A -85,B 0,C 180,E1 32344.444,E2 32344.444} C_VEL
LIN {X 0,Y 717.941,Z 960.708,A -85,B 0,C 180,E1 32343.518,E2 32343.518} C_VEL
LIN {X 0,Y 717.25,Z 982.995,A -85,B 0,C 180,E1 32342.412,E2 32342.412} C_VEL
LIN {X 0,Y 716.464,Z 1007.894,A -85,B 0,C 180,E1 32340.994,E2 32340.994} C_VEL
LIN {X 0,Y 715.787,Z 1027.578,A -85,B 0,C 180,E1 32339.728,E2 32339.728} C_VEL
LIN {X 0,Y 715.19,Z 1045.813,A -85,B 0,C 180,E1 32338.431,E2 32338.431} C_VEL
LIN {X 0,Y 714.548,Z 1067.22,A -85,B 0,C 180,E1 32336.735,E2 32336.735} C_VEL
LIN {X 0,Y 713.971,Z 1085.454,A -85,B 0,C 180,E1 32335.108,E2 32335.108} C_VEL
LIN {X 0,Y 713.51,Z 1101.398,A -85,B 0,C 180,E1 32333.539,E2 32333.539} C_VEL
LIN {X 0,Y 713.048,Z 1120.128,A -85,B 0,C 180,E1 32331.468,E2 32331.468} C_VEL
LIN {X 0,Y 712.741,Z 1134.092,A -85,B 0,C 180,E1 32329.723,E2 32329.723} C_VEL
LIN {X 0,Y 712.497,Z 1146.006,A -85,B 0,C 180,E1 32328.067,E2 32328.067} C_VEL
LIN {X 0,Y 712.28,Z 1158.901,A -85,B 0,C 180,E1 32326.054,E2 32326.054} C_VEL
LIN {X 0,Y 712.124,Z 1170.245,A -85,B 0,C 180,E1 32323.975,E2 32323.975} C_VEL
LIN {X 0,Y 712.027,Z 1178.434,A -85,B 0,C 180,E1 32322.242,E2 32322.242} C_VEL
LIN {X 0,Y 711.98,Z 1186.134,A -85,B 0,C 180,E1 32320.355,E2 32320.355} C_VEL
LIN {X 0,Y 711.935,Z 1193.355,A -85,B 0,C 180,E1 32318.155,E2 32318.155} C_VEL
LIN {X 0,Y 711.916,Z 1198.765,A -85,B 0,C 180,E1 32315.965,E2 32315.965} C_VEL
LIN {X 0,Y 711.907,Z 1202.382,A -85,B 0,C 180,E1 32313.865,E2 32313.865} C_VEL
LIN {X 0,Y 711.909,Z 1204.549,A -85,B 0,C 180,E1 32311.61,E2 32311.61} C_VEL
LIN {X 0,Y 711.89,Z 1204.872,A -85,B 0,C 180,E1 32309.517,E2 32309.517} C_VEL
LIN {X 0,Y 711.907,Z 1203.967,A -85,B 0,C 180,E1 32307.585,E2 32307.585} C_VEL
LIN {X 0,Y 711.908,Z 1201.303,A -85,B 0,C 180,E1 32305.408,E2 32305.408} C_VEL
LIN {X 0,Y 711.919,Z 1197.152,A -85,B 0,C 180,E1 32303.306,E2 32303.306} C_VEL
LIN {X 0,Y 711.945,Z 1191.397,A -85,B 0,C 180,E1 32301.195,E2 32301.195} C_VEL
LIN {X 0,Y 711.977,Z 1183.958,A -85,B 0,C 180,E1 32299.071,E2 32299.071} C_VEL
LIN {X 0,Y 712.09,Z 1173.94,A -85,B 0,C 180,E1 32296.769,E2 32296.769} C_VEL
LIN {X 0,Y 712.178,Z 1164.531,A -85,B 0,C 180,E1 32294.946,E2 32294.946} C_VEL
LIN {X 0,Y 712.341,Z 1154.745,A -85,B 0,C 180,E1 32293.277,E2 32293.277} C_VEL
LIN {X 0,Y 712.542,Z 1143.678,A -85,B 0,C 180,E1 32291.595,E2 32291.595} C_VEL
LIN {X 0,Y 712.858,Z 1129.296,A -85,B 0,C 180,E1 32289.644,E2 32289.644} C_VEL
LIN {X 0,Y 713.224,Z 1112.625,A -85,B 0,C 180,E1 32287.672,E2 32287.672} C_VEL
LIN {X 0,Y 713.611,Z 1097.983,A -85,B 0,C 180,E1 32286.114,E2 32286.114} C_VEL
LIN {X 0,Y 714.174,Z 1079.334,A -85,B 0,C 180,E1 32284.317,E2 32284.317} C_VEL
LIN {X 0,Y 714.745,Z 1059.886,A -85,B 0,C 180,E1 32282.665,E2 32282.665} C_VEL
LIN {X 0,Y 715.326,Z 1042.24,A -85,B 0,C 180,E1 32281.306,E2 32281.306} C_VEL
LIN {X 0,Y 716.075,Z 1020.251,A -85,B 0,C 180,E1 32279.777,E2 32279.777} C_VEL
LIN {X 0,Y 716.773,Z 997.046,A -85,B 0,C 180,E1 32278.366,E2 32278.366} C_VEL
LIN {X 0,Y 717.451,Z 976.762,A -85,B 0,C 180,E1 32277.267,E2 32277.267} C_VEL
LIN {X 0,Y 718.191,Z 954.383,A -85,B 0,C 180,E1 32276.192,E2 32276.192} C_VEL
LIN {X 0,Y 718.939,Z 927.689,A -85,B 0,C 180,E1 32275.09,E2 32275.09} C_VEL
LIN {X 0,Y 719.505,Z 905.599,A -85,B 0,C 180,E1 32274.317,E2 32274.317} C_VEL
LIN {X 0,Y 720.071,Z 882.549,A -85,B 0,C 180,E1 32273.63,E2 32273.63} C_VEL
LIN {X 0,Y 720.646,Z 855.599,A -85,B 0,C 180,E1 32272.99,E2 32272.99} C_VEL
LIN {X 0,Y 721.041,Z 828.401,A -85,B 0,C 180,E1 32272.512,E2 32272.512} C_VEL
LIN {X 0,Y 722.488,Z 599.457,A -85,B 0,C 180,E1 32269.713,E2 32269.713} C_VEL
LIN {X 0,Y 723.793,Z 395.011,A -85,B 0,C 180,E1 32267.146,E2 32267.146} C_VEL
LIN {X 0,Y 723.842,Z 363.09,A -85,B 0,C 180,E1 32266.725,E2 32266.725} C_VEL
LIN {X 0,Y 720.488,Z 350.376,A -85,B 0,C 180,E1 32266.283,E2 32266.283} C_VEL
LIN {X 0,Y 720.466,Z 344.152,A -85,B 0,C 180,E1 32265.84,E2 32265.84} C_VEL
LIN {X 0,Y 713.808,Z 329.349,A -85,B 0,C 180,E1 32264.234,E2 32264.234} C_VEL
LIN {X 0,Y 712.26,Z 325.854,A -85,B 0,C 180,E1 32263.846,E2 32263.846} C_VEL
LIN {X 0,Y 712.207,Z 325.517,A -85,B 0,C 180,E1 32263.8,E2 32263.8} C_VEL
LIN {X 0,Y 712.206,Z 325.513,A -85,B 0,C 180,E1 32261.289,E2 32261.289} C_VEL
LIN {X 0,Y 712.285,Z 325.51,A -85,B 0,C 180,E1 32258.438,E2 32258.438} C_VEL
LIN {X 0,Y 712.208,Z 325.512,A -85,B 0,C 180,E1 32255.537,E2 32255.537} C_VEL
LIN {X 0,Y 712.211,Z 325.508,A -85,B 0,C 180,E1 32253.006,E2 32253.006} C_VEL
LIN {X 0,Y 712.287,Z 325.501,A -85,B 0,C 180,E1 32250.076,E2 32250.076} C_VEL
LIN {X 0,Y 712.206,Z 325.498,A -85,B 0,C 180,E1 32247.238,E2 32247.238} C_VEL
LIN {X 0,Y 712.215,Z 325.508,A -85,B 0,C 180,E1 32244.728,E2 32244.728} C_VEL
LIN {X 0,Y 712.278,Z 325.499,A -85,B 0,C 180,E1 32241.753,E2 32241.753} C_VEL
LIN {X 0,Y 712.209,Z 325.506,A -85,B 0,C 180,E1 32239.009,E2 32239.009} C_VEL
LIN {X 0,Y 712.217,Z 325.5,A -85,B 0,C 180,E1 32236.475,E2 32236.475} C_VEL
LIN {X 0,Y 712.282,Z 325.504,A -85,B 0,C 180,E1 32233.558,E2 32233.558} C_VEL
LIN {X 0,Y 712.211,Z 325.507,A -85,B 0,C 180,E1 32230.762,E2 32230.762} C_VEL
LIN {X 0,Y 712.226,Z 325.504,A -85,B 0,C 180,E1 32228.152,E2 32228.152} C_VEL
LIN {X 0,Y 712.266,Z 325.508,A -85,B 0,C 180,E1 32225.155,E2 32225.155} C_VEL
LIN {X 0,Y 712.21,Z 325.502,A -85,B 0,C 180,E1 32222.414,E2 32222.414} C_VEL
LIN {X 0,Y 712.243,Z 325.5,A -85,B 0,C 180,E1 32219.759,E2 32219.759} C_VEL
LIN {X 0,Y 712.24,Z 325.499,A -85,B 0,C 180,E1 32216.7,E2 32216.7} C_VEL
LIN {X 0,Y 712.214,Z 325.506,A -85,B 0,C 180,E1 32214.037,E2 32214.037} C_VEL
LIN {X 0,Y 712.276,Z 325.501,A -85,B 0,C 180,E1 32211.28,E2 32211.28} C_VEL
LIN {X 0,Y 712.225,Z 325.51,A -85,B 0,C 180,E1 32208.254,E2 32208.254} C_VEL
LIN {X 0,Y 712.221,Z 325.496,A -85,B 0,C 180,E1 32205.612,E2 32205.612} C_VEL
LIN {X 0,Y 712.283,Z 325.509,A -85,B 0,C 180,E1 32202.657,E2 32202.657} C_VEL
LIN {X 0,Y 712.281,Z 325.498,A -85,B 0,C 180,E1 32200.812,E2 32200.812} C_VEL
LIN {X 0,Y 711.298,Z 325.623,A -85,B 0,C 180,E1 32200.192,E2 32200.192} C_VEL
LIN {X 0,Y 704.85,Z 326.436,A -85,B 0,C 180,E1 32198.457,E2 32198.457} C_VEL
LIN {X 0,Y 704.292,Z 326.497,A -85,B 0,C 180,E1 32198.005,E2 32198.005} C_VEL
LIN {X 0,Y 704.285,Z 326.492,A -85,B 0,C 180,E1 32195.329,E2 32195.329} C_VEL
LIN {X 0,Y 704.343,Z 326.498,A -85,B 0,C 180,E1 32192.341,E2 32192.341} C_VEL
LIN {X 0,Y 704.282,Z 326.497,A -85,B 0,C 180,E1 32189.513,E2 32189.513} C_VEL
LIN {X 0,Y 704.318,Z 326.496,A -85,B 0,C 180,E1 32186.771,E2 32186.771} C_VEL
LIN {X 0,Y 704.306,Z 326.502,A -85,B 0,C 180,E1 32183.7,E2 32183.7} C_VEL
LIN {X 0,Y 704.322,Z 326.736,A -85,B 0,C 180,E1 32182.991,E2 32182.991} C_VEL
LIN {X 0,Y 705.508,Z 329.808,A -85,B 0,C 180,E1 32182.657,E2 32182.657} C_VEL
LIN {X 0,Y 710.74,Z 341.272,A -85,B 0,C 180,E1 32181.396,E2 32181.396} C_VEL
LIN {X 0,Y 716.409,Z 349.938,A -85,B 0,C 180,E1 32180.835,E2 32180.835} C_VEL
LIN {X 0,Y 718.17,Z 357.096,A -85,B 0,C 180,E1 32180.603,E2 32180.603} C_VEL
LIN {X 0,Y 716.549,Z 566.305,A -85,B 0,C 180,E1 32177.946,E2 32177.946} C_VEL
LIN {X 0,Y 714.967,Z 789.787,A -85,B 0,C 180,E1 32175.199,E2 32175.199} C_VEL
LIN {X 0,Y 714.586,Z 825.441,A -85,B 0,C 180,E1 32174.727,E2 32174.727} C_VEL
LIN {X 0,Y 714.033,Z 851.913,A -85,B 0,C 180,E1 32174.218,E2 32174.218} C_VEL
LIN {X 0,Y 713.456,Z 877.327,A -85,B 0,C 180,E1 32173.581,E2 32173.581} C_VEL
LIN {X 0,Y 712.698,Z 904.09,A -85,B 0,C 180,E1 32172.739,E2 32172.739} C_VEL
LIN {X 0,Y 711.868,Z 929.045,A -85,B 0,C 180,E1 32171.794,E2 32171.794} C_VEL
LIN {X 0,Y 711.027,Z 951.998,A -85,B 0,C 180,E1 32170.782,E2 32170.782} C_VEL
LIN {X 0,Y 710.123,Z 976.756,A -85,B 0,C 180,E1 32169.525,E2 32169.525} C_VEL
LIN {X 0,Y 709.243,Z 999.747,A -85,B 0,C 180,E1 32168.183,E2 32168.183} C_VEL
LIN {X 0,Y 708.343,Z 1022.284,A -85,B 0,C 180,E1 32166.699,E2 32166.699} C_VEL
LIN {X 0,Y 707.51,Z 1044.856,A -85,B 0,C 180,E1 32165.013,E2 32165.013} C_VEL
LIN {X 0,Y 706.721,Z 1065.636,A -85,B 0,C 180,E1 32163.262,E2 32163.262} C_VEL
LIN {X 0,Y 706.038,Z 1086.087,A -85,B 0,C 180,E1 32161.314,E2 32161.314} C_VEL
LIN {X 0,Y 705.482,Z 1103.383,A -85,B 0,C 180,E1 32159.458,E2 32159.458} C_VEL
LIN {X 0,Y 705.01,Z 1120.743,A -85,B 0,C 180,E1 32157.355,E2 32157.355} C_VEL
LIN {X 0,Y 704.65,Z 1134.438,A -85,B 0,C 180,E1 32155.464,E2 32155.464} C_VEL
LIN {X 0,Y 704.386,Z 1146.458,A -85,B 0,C 180,E1 32153.596,E2 32153.596} C_VEL
LIN {X 0,Y 704.198,Z 1158.739,A -85,B 0,C 180,E1 32151.401,E2 32151.401} C_VEL
LIN {X 0,Y 704.047,Z 1168.51,A -85,B 0,C 180,E1 32149.323,E2 32149.323} C_VEL
LIN {X 0,Y 703.988,Z 1176.09,A -85,B 0,C 180,E1 32147.438,E2 32147.438} C_VEL
LIN {X 0,Y 703.942,Z 1183.003,A -85,B 0,C 180,E1 32145.319,E2 32145.319} C_VEL
LIN {X 0,Y 703.922,Z 1188.284,A -85,B 0,C 180,E1 32143.22,E2 32143.22} C_VEL
LIN {X 0,Y 703.911,Z 1192.165,A -85,B 0,C 180,E1 32141.021,E2 32141.021} C_VEL
LIN {X 0,Y 703.907,Z 1194.382,A -85,B 0,C 180,E1 32138.824,E2 32138.824} C_VEL
LIN {X 0,Y 703.903,Z 1194.889,A -85,B 0,C 180,E1 32136.525,E2 32136.525} C_VEL
LIN {X 0,Y 703.907,Z 1193.94,A -85,B 0,C 180,E1 32134.481,E2 32134.481} C_VEL
LIN {X 0,Y 703.915,Z 1191.258,A -85,B 0,C 180,E1 32132.279,E2 32132.279} C_VEL
LIN {X 0,Y 703.929,Z 1187.041,A -85,B 0,C 180,E1 32130.14,E2 32130.14} C_VEL
LIN {X 0,Y 703.961,Z 1181.139,A -85,B 0,C 180,E1 32127.965,E2 32127.965} C_VEL
LIN {X 0,Y 704.032,Z 1173.123,A -85,B 0,C 180,E1 32125.683,E2 32125.683} C_VEL
LIN {X 0,Y 704.121,Z 1163.489,A -85,B 0,C 180,E1 32123.477,E2 32123.477} C_VEL
LIN {X 0,Y 704.271,Z 1153.792,A -85,B 0,C 180,E1 32121.592,E2 32121.592} C_VEL
LIN {X 0,Y 704.503,Z 1142.152,A -85,B 0,C 180,E1 32119.616,E2 32119.616} C_VEL
LIN {X 0,Y 704.83,Z 1126.943,A -85,B 0,C 180,E1 32117.381,E2 32117.381} C_VEL
LIN {X 0,Y 705.217,Z 1112.014,A -85,B 0,C 180,E1 32115.466,E2 32115.466} C_VEL
LIN {X 0,Y 705.737,Z 1095.176,A -85,B 0,C 180,E1 32113.54,E2 32113.54} C_VEL
LIN {X 0,Y 706.342,Z 1076.811,A -85,B 0,C 180,E1 32111.685,E2 32111.685} C_VEL
LIN {X 0,Y 707.035,Z 1057.107,A -85,B 0,C 180,E1 32109.901,E2 32109.901} C_VEL
LIN {X 0,Y 707.845,Z 1035.723,A -85,B 0,C 180,E1 32108.192,E2 32108.192} C_VEL
LIN {X 0,Y 708.694,Z 1014.006,A -85,B 0,C 180,E1 32106.644,E2 32106.644} C_VEL
LIN {X 0,Y 709.623,Z 989.115,A -85,B 0,C 180,E1 32105.084,E2 32105.084} C_VEL
LIN {X 0,Y 710.528,Z 966.07,A -85,B 0,C 180,E1 32103.822,E2 32103.822} C_VEL
LIN {X 0,Y 711.42,Z 942.288,A -85,B 0,C 180,E1 32102.681,E2 32102.681} C_VEL
LIN {X 0,Y 712.242,Z 916.729,A -85,B 0,C 180,E1 32101.628,E2 32101.628} C_VEL
LIN {X 0,Y 713.003,Z 891.898,A -85,B 0,C 180,E1 32100.767,E2 32100.767} C_VEL
LIN {X 0,Y 713.694,Z 867.14,A -85,B 0,C 180,E1 32100.057,E2 32100.057} C_VEL
LIN {X 0,Y 714.31,Z 840.283,A -85,B 0,C 180,E1 32099.448,E2 32099.448} C_VEL
LIN {X 0,Y 714.746,Z 813.935,A -85,B 0,C 180,E1 32099.012,E2 32099.012} C_VEL
LIN {X 0,Y 716.384,Z 588.489,A -85,B 0,C 180,E1 32096.241,E2 32096.241} C_VEL
LIN {X 0,Y 717.989,Z 377.087,A -85,B 0,C 180,E1 32093.563,E2 32093.563} C_VEL
LIN {X 0,Y 717.992,Z 355.942,A -85,B 0,C 180,E1 32093.278,E2 32093.278} C_VEL
LIN {X 0,Y 715.911,Z 349.087,A -85,B 0,C 180,E1 32093.025,E2 32093.025} C_VEL
LIN {X 0,Y 710.212,Z 340.393,A -85,B 0,C 180,E1 32092.433,E2 32092.433} C_VEL
LIN {X 0,Y 705.791,Z 330.319,A -85,B 0,C 180,E1 32091.316,E2 32091.316} C_VEL
LIN {X 0,Y 704.287,Z 326.862,A -85,B 0,C 180,E1 32090.925,E2 32090.925} C_VEL
LIN {X 0,Y 704.238,Z 326.508,A -85,B 0,C 180,E1 32090.817,E2 32090.817} C_VEL
LIN {X 0,Y 704.278,Z 326.504,A -85,B 0,C 180,E1 32088.254,E2 32088.254} C_VEL
LIN {X 0,Y 704.258,Z 326.504,A -85,B 0,C 180,E1 32085.226,E2 32085.226} C_VEL
LIN {X 0,Y 704.237,Z 326.497,A -85,B 0,C 180,E1 32082.74,E2 32082.74} C_VEL
LIN {X 0,Y 704.248,Z 326.502,A -85,B 0,C 180,E1 32080.348,E2 32080.348} C_VEL
LIN {X 0,Y 704.316,Z 326.498,A -85,B 0,C 180,E1 32077.418,E2 32077.418} C_VEL
LIN {X 0,Y 704.244,Z 326.497,A -85,B 0,C 180,E1 32074.705,E2 32074.705} C_VEL
LIN {X 0,Y 704.241,Z 326.5,A -85,B 0,C 180,E1 32072.354,E2 32072.354} C_VEL
LIN {X 0,Y 704.279,Z 326.502,A -85,B 0,C 180,E1 32069.796,E2 32069.796} C_VEL
LIN {X 0,Y 704.265,Z 326.495,A -85,B 0,C 180,E1 32066.747,E2 32066.747} C_VEL
LIN {X 0,Y 704.243,Z 326.5,A -85,B 0,C 180,E1 32064.289,E2 32064.289} C_VEL
LIN {X 0,Y 704.255,Z 326.488,A -85,B 0,C 180,E1 32061.838,E2 32061.838} C_VEL
LIN {X 0,Y 704.315,Z 326.499,A -85,B 0,C 180,E1 32058.886,E2 32058.886} C_VEL
LIN {X 0,Y 704.246,Z 326.498,A -85,B 0,C 180,E1 32056.158,E2 32056.158} C_VEL
LIN {X 0,Y 704.248,Z 326.499,A -85,B 0,C 180,E1 32053.8,E2 32053.8} C_VEL
LIN {X 0,Y 704.322,Z 326.501,A -85,B 0,C 180,E1 32051.049,E2 32051.049} C_VEL
LIN {X 0,Y 704.261,Z 326.499,A -85,B 0,C 180,E1 32048.162,E2 32048.162} C_VEL
LIN {X 0,Y 704.247,Z 326.496,A -85,B 0,C 180,E1 32045.786,E2 32045.786} C_VEL
LIN {X 0,Y 704.261,Z 326.5,A -85,B 0,C 180,E1 32043.337,E2 32043.337} C_VEL
LIN {X 0,Y 704.309,Z 326.495,A -85,B 0,C 180,E1 32040.325,E2 32040.325} C_VEL
LIN {X 0,Y 704.251,Z 326.499,A -85,B 0,C 180,E1 32037.64,E2 32037.64} C_VEL
LIN {X 0,Y 704.257,Z 326.495,A -85,B 0,C 180,E1 32035.195,E2 32035.195} C_VEL
LIN {X 0,Y 704.333,Z 326.494,A -85,B 0,C 180,E1 32032.249,E2 32032.249} C_VEL
LIN {X 0,Y 704.254,Z 326.497,A -85,B 0,C 180,E1 32029.447,E2 32029.447} C_VEL
LIN {X 0,Y 704.256,Z 326.483,A -85,B 0,C 180,E1 32027.037,E2 32027.037} C_VEL
LIN {X 0,Y 704.345,Z 326.499,A -85,B 0,C 180,E1 32024.183,E2 32024.183} C_VEL
LIN {X 0,Y 704.257,Z 326.484,A -85,B 0,C 180,E1 32021.284,E2 32021.284} C_VEL
LIN {X 0,Y 704.257,Z 326.497,A -85,B 0,C 180,E1 32018.861,E2 32018.861} C_VEL
LIN {X 0,Y 704.333,Z 326.485,A -85,B 0,C 180,E1 32016.093,E2 32016.093} C_VEL
LIN {X 0,Y 704.265,Z 326.498,A -85,B 0,C 180,E1 32013.161,E2 32013.161} C_VEL
LIN {X 0,Y 704.257,Z 326.498,A -85,B 0,C 180,E1 32010.764,E2 32010.764} C_VEL
LIN {X 0,Y 704.3,Z 326.499,A -85,B 0,C 180,E1 32008.121,E2 32008.121} C_VEL
LIN {X 0,Y 704.28,Z 326.499,A -85,B 0,C 180,E1 32005.099,E2 32005.099} C_VEL
LIN {X 0,Y 704.259,Z 326.501,A -85,B 0,C 180,E1 32002.526,E2 32002.526} C_VEL
LIN {X 0,Y 704.306,Z 326.504,A -85,B 0,C 180,E1 31999.869,E2 31999.869} C_VEL
LIN {X 0,Y 704.278,Z 326.505,A -85,B 0,C 180,E1 31996.818,E2 31996.818} C_VEL
LIN {X 0,Y 705.678,Z 330.148,A -85,B 0,C 180,E1 31996.387,E2 31996.387} C_VEL
LIN {X 0,Y 711.7,Z 343.187,A -85,B 0,C 180,E1 31994.92,E2 31994.92} C_VEL
LIN {X 0,Y 714.114,Z 348.876,A -85,B 0,C 180,E1 31994.316,E2 31994.316} C_VEL
LIN {X 0,Y 714.219,Z 351.372,A -85,B 0,C 180,E1 31994.167,E2 31994.167} C_VEL
LIN {X 0,Y 718.152,Z 366.631,A -85,B 0,C 180,E1 31993.656,E2 31993.656} C_VEL
LIN {X 0,Y 716.539,Z 577.786,A -85,B 0,C 180,E1 31990.972,E2 31990.972} C_VEL
LIN {X 0,Y 714.955,Z 801.663,A -85,B 0,C 180,E1 31988.221,E2 31988.221} C_VEL
LIN {X 0,Y 714.579,Z 836.005,A -85,B 0,C 180,E1 31987.763,E2 31987.763} C_VEL
LIN {X 0,Y 714.009,Z 863.174,A -85,B 0,C 180,E1 31987.235,E2 31987.235} C_VEL
LIN {X 0,Y 713.419,Z 888.318,A -85,B 0,C 180,E1 31986.597,E2 31986.597} C_VEL
LIN {X 0,Y 712.626,Z 916.206,A -85,B 0,C 180,E1 31985.709,E2 31985.709} C_VEL
LIN {X 0,Y 711.838,Z 939.506,A -85,B 0,C 180,E1 31984.818,E2 31984.818} C_VEL
LIN {X 0,Y 711.07,Z 960.711,A -85,B 0,C 180,E1 31983.885,E2 31983.885} C_VEL
LIN {X 0,Y 710.257,Z 982.228,A -85,B 0,C 180,E1 31982.812,E2 31982.812} C_VEL
LIN {X 0,Y 709.316,Z 1007.891,A -85,B 0,C 180,E1 31981.342,E2 31981.342} C_VEL
LIN {X 0,Y 708.531,Z 1027.58,A -85,B 0,C 180,E1 31980.064,E2 31980.064} C_VEL
LIN {X 0,Y 707.805,Z 1046.476,A -85,B 0,C 180,E1 31978.704,E2 31978.704} C_VEL
LIN {X 0,Y 706.984,Z 1068.744,A -85,B 0,C 180,E1 31976.908,E2 31976.908} C_VEL
LIN {X 0,Y 706.367,Z 1085.921,A -85,B 0,C 180,E1 31975.352,E2 31975.352} C_VEL
LIN {X 0,Y 705.803,Z 1102.248,A -85,B 0,C 180,E1 31973.723,E2 31973.723} C_VEL
LIN {X 0,Y 705.276,Z 1120.13,A -85,B 0,C 180,E1 31971.716,E2 31971.716} C_VEL
LIN {X 0,Y 704.918,Z 1133.811,A -85,B 0,C 180,E1 31969.989,E2 31969.989} C_VEL
LIN {X 0,Y 704.607,Z 1146.59,A -85,B 0,C 180,E1 31968.191,E2 31968.191} C_VEL
LIN {X 0,Y 704.335,Z 1160.068,A -85,B 0,C 180,E1 31966.036,E2 31966.036} C_VEL
LIN {X 0,Y 704.164,Z 1170.657,A -85,B 0,C 180,E1 31964.052,E2 31964.052} C_VEL
LIN {X 0,Y 704.053,Z 1178.792,A -85,B 0,C 180,E1 31962.299,E2 31962.299} C_VEL
LIN {X 0,Y 703.99,Z 1186.427,A -85,B 0,C 180,E1 31960.392,E2 31960.392} C_VEL
LIN {X 0,Y 703.94,Z 1193.595,A -85,B 0,C 180,E1 31958.166,E2 31958.166} C_VEL
LIN {X 0,Y 703.918,Z 1198.937,A -85,B 0,C 180,E1 31955.952,E2 31955.952} C_VEL
LIN {X 0,Y 703.908,Z 1202.484,A -85,B 0,C 180,E1 31953.828,E2 31953.828} C_VEL
LIN {X 0,Y 703.908,Z 1204.549,A -85,B 0,C 180,E1 31951.628,E2 31951.628} C_VEL
LIN {X 0,Y 703.89,Z 1204.872,A -85,B 0,C 180,E1 31949.512,E2 31949.512} C_VEL
LIN {X 0,Y 703.907,Z 1203.964,A -85,B 0,C 180,E1 31947.558,E2 31947.558} C_VEL
LIN {X 0,Y 703.909,Z 1201.428,A -85,B 0,C 180,E1 31945.438,E2 31945.438} C_VEL
LIN {X 0,Y 703.921,Z 1197.348,A -85,B 0,C 180,E1 31943.311,E2 31943.311} C_VEL
LIN {X 0,Y 703.949,Z 1191.394,A -85,B 0,C 180,E1 31941.094,E2 31941.094} C_VEL
LIN {X 0,Y 703.992,Z 1184.277,A -85,B 0,C 180,E1 31939.029,E2 31939.029} C_VEL
LIN {X 0,Y 704.128,Z 1173.941,A -85,B 0,C 180,E1 31936.617,E2 31936.617} C_VEL
LIN {X 0,Y 704.237,Z 1164.533,A -85,B 0,C 180,E1 31934.772,E2 31934.772} C_VEL
LIN {X 0,Y 704.437,Z 1154.7,A -85,B 0,C 180,E1 31933.076,E2 31933.076} C_VEL
LIN {X 0,Y 704.667,Z 1143.68,A -85,B 0,C 180,E1 31931.382,E2 31931.382} C_VEL
LIN {X 0,Y 705.06,Z 1128.62,A -85,B 0,C 180,E1 31929.322,E2 31929.322} C_VEL
LIN {X 0,Y 705.487,Z 1112.627,A -85,B 0,C 180,E1 31927.414,E2 31927.414} C_VEL
LIN {X 0,Y 705.973,Z 1097.612,A -85,B 0,C 180,E1 31925.8,E2 31925.8} C_VEL
LIN {X 0,Y 706.607,Z 1078.762,A -85,B 0,C 180,E1 31923.97,E2 31923.97} C_VEL
LIN {X 0,Y 707.314,Z 1059.614,A -85,B 0,C 180,E1 31922.331,E2 31922.331} C_VEL
LIN {X 0,Y 707.954,Z 1042.846,A -85,B 0,C 180,E1 31921.025,E2 31921.025} C_VEL
LIN {X 0,Y 708.73,Z 1022.922,A -85,B 0,C 180,E1 31919.618,E2 31919.618} C_VEL
LIN {X 0,Y 709.633,Z 998.654,A -85,B 0,C 180,E1 31918.105,E2 31918.105} C_VEL
LIN {X 0,Y 710.413,Z 978.546,A -85,B 0,C 180,E1 31916.998,E2 31916.998} C_VEL
LIN {X 0,Y 711.154,Z 958.824,A -85,B 0,C 180,E1 31916.027,E2 31916.027} C_VEL
LIN {X 0,Y 711.932,Z 937.251,A -85,B 0,C 180,E1 31915.089,E2 31915.089} C_VEL
LIN {X 0,Y 712.777,Z 911.467,A -85,B 0,C 180,E1 31914.126,E2 31914.126} C_VEL
LIN {X 0,Y 713.471,Z 885.657,A -85,B 0,C 180,E1 31913.329,E2 31913.329} C_VEL
LIN {X 0,Y 714.088,Z 860.466,A -85,B 0,C 180,E1 31912.705,E2 31912.705} C_VEL
LIN {X 0,Y 714.616,Z 832.883,A -85,B 0,C 180,E1 31912.187,E2 31912.187} C_VEL
LIN {X 0,Y 715.061,Z 786.137,A -85,B 0,C 180,E1 31911.591,E2 31911.591} C_VEL
LIN {X 0,Y 716.677,Z 560.283,A -85,B 0,C 180,E1 31908.809,E2 31908.809} C_VEL
LIN {X 0,Y 718.157,Z 365.917,A -85,B 0,C 180,E1 31906.335,E2 31906.335} C_VEL
LIN {X 0,Y 714.069,Z 350.376,A -85,B 0,C 180,E1 31905.788,E2 31905.788} C_VEL
LIN {X 0,Y 713.999,Z 348.337,A -85,B 0,C 180,E1 31905.636,E2 31905.636} C_VEL
LIN {X 0,Y 707.481,Z 334.008,A -85,B 0,C 180,E1 31904.055,E2 31904.055} C_VEL
LIN {X 0,Y 704.357,Z 327.035,A -85,B 0,C 180,E1 31903.263,E2 31903.263} C_VEL
LIN {X 0,Y 704.279,Z 326.505,A -85,B 0,C 180,E1 31903.182,E2 31903.182} C_VEL
LIN {X 0,Y 704.316,Z 326.503,A -85,B 0,C 180,E1 31900.13,E2 31900.13} C_VEL
LIN {X 0,Y 704.264,Z 326.501,A -85,B 0,C 180,E1 31897.421,E2 31897.421} C_VEL
LIN {X 0,Y 704.294,Z 326.498,A -85,B 0,C 180,E1 31894.801,E2 31894.801} C_VEL
LIN {X 0,Y 704.289,Z 326.487,A -85,B 0,C 180,E1 31891.688,E2 31891.688} C_VEL
LIN {X 0,Y 704.266,Z 326.498,A -85,B 0,C 180,E1 31889.142,E2 31889.142} C_VEL
LIN {X 0,Y 704.305,Z 326.482,A -85,B 0,C 180,E1 31886.473,E2 31886.473} C_VEL
LIN {X 0,Y 704.29,Z 326.49,A -85,B 0,C 180,E1 31883.423,E2 31883.423} C_VEL
LIN {X 0,Y 704.268,Z 326.496,A -85,B 0,C 180,E1 31880.877,E2 31880.877} C_VEL
LIN {X 0,Y 704.312,Z 326.491,A -85,B 0,C 180,E1 31878.2,E2 31878.2} C_VEL
LIN {X 0,Y 704.287,Z 326.5,A -85,B 0,C 180,E1 31875.122,E2 31875.122} C_VEL
LIN {X 0,Y 704.27,Z 326.485,A -85,B 0,C 180,E1 31872.546,E2 31872.546} C_VEL
LIN {X 0,Y 704.343,Z 326.492,A -85,B 0,C 180,E1 31869.726,E2 31869.726} C_VEL
LIN {X 0,Y 704.279,Z 326.487,A -85,B 0,C 180,E1 31866.767,E2 31866.767} C_VEL
LIN {X 0,Y 704.28,Z 326.496,A -85,B 0,C 180,E1 31864.152,E2 31864.152} C_VEL
LIN {X 0,Y 704.344,Z 326.483,A -85,B 0,C 180,E1 31861.22,E2 31861.22} C_VEL
LIN {X 0,Y 704.275,Z 326.498,A -85,B 0,C 180,E1 31858.373,E2 31858.373} C_VEL
LIN {X 0,Y 704.299,Z 326.481,A -85,B 0,C 180,E1 31855.685,E2 31855.685} C_VEL
LIN {X 0,Y 704.304,Z 326.497,A -85,B 0,C 180,E1 31852.577,E2 31852.577} C_VEL
LIN {X 0,Y 704.276,Z 326.488,A -85,B 0,C 180,E1 31849.943,E2 31849.943} C_VEL
LIN {X 0,Y 704.339,Z 326.493,A -85,B 0,C 180,E1 31847.122,E2 31847.122} C_VEL
LIN {X 0,Y 704.292,Z 326.498,A -85,B 0,C 180,E1 31844.182,E2 31844.182} C_VEL
LIN {X 0,Y 704.284,Z 326.49,A -85,B 0,C 180,E1 31841.504,E2 31841.504} C_VEL
LIN {X 0,Y 704.343,Z 326.497,A -85,B 0,C 180,E1 31838.515,E2 31838.515} C_VEL
LIN {X 0,Y 704.292,Z 326.497,A -85,B 0,C 180,E1 31838.005,E2 31838.005} C_VEL
LIN {X 0,Y 703.269,Z 326.62,A -85,B 0,C 180,E1 31837.379,E2 31837.379} C_VEL
LIN {X 0,Y 696.856,Z 327.418,A -85,B 0,C 180,E1 31835.622,E2 31835.622} C_VEL
LIN {X 0,Y 696.357,Z 327.48,A -85,B 0,C 180,E1 31835.166,E2 31835.166} C_VEL
LIN {X 0,Y 696.383,Z 327.49,A -85,B 0,C 180,E1 31832.09,E2 31832.09} C_VEL
LIN {X 0,Y 696.343,Z 327.485,A -85,B 0,C 180,E1 31829.326,E2 31829.326} C_VEL
LIN {X 0,Y 696.405,Z 327.487,A -85,B 0,C 180,E1 31826.442,E2 31826.442} C_VEL
LIN {X 0,Y 696.379,Z 327.635,A -85,B 0,C 180,E1 31823.602,E2 31823.602} C_VEL
LIN {X 0,Y 697.787,Z 331.173,A -85,B 0,C 180,E1 31823.204,E2 31823.204} C_VEL
LIN {X 0,Y 702.425,Z 341.29,A -85,B 0,C 180,E1 31822.065,E2 31822.065} C_VEL
LIN {X 0,Y 711.295,Z 354.653,A -85,B 0,C 180,E1 31821.167,E2 31821.167} C_VEL
LIN {X 0,Y 712.35,Z 359.301,A -85,B 0,C 180,E1 31821.021,E2 31821.021} C_VEL
LIN {X 0,Y 710.486,Z 568.11,A -85,B 0,C 180,E1 31818.348,E2 31818.348} C_VEL
LIN {X 0,Y 708.664,Z 791.65,A -85,B 0,C 180,E1 31815.578,E2 31815.578} C_VEL
LIN {X 0,Y 708.226,Z 826.032,A -85,B 0,C 180,E1 31815.116,E2 31815.116} C_VEL
LIN {X 0,Y 707.608,Z 852.278,A -85,B 0,C 180,E1 31814.606,E2 31814.606} C_VEL
LIN {X 0,Y 706.934,Z 877.759,A -85,B 0,C 180,E1 31813.962,E2 31813.962} C_VEL
LIN {X 0,Y 706.048,Z 904.827,A -85,B 0,C 180,E1 31813.101,E2 31813.101} C_VEL
LIN {X 0,Y 705.14,Z 929.067,A -85,B 0,C 180,E1 31812.175,E2 31812.175} C_VEL
LIN {X 0,Y 704.185,Z 952.007,A -85,B 0,C 180,E1 31811.156,E2 31811.156} C_VEL
LIN {X 0,Y 703.115,Z 976.732,A -85,B 0,C 180,E1 31809.892,E2 31809.892} C_VEL
LIN {X 0,Y 702.12,Z 999.658,A -85,B 0,C 180,E1 31808.542,E2 31808.542} C_VEL
LIN {X 0,Y 701.058,Z 1022.944,A -85,B 0,C 180,E1 31806.993,E2 31806.993} C_VEL
LIN {X 0,Y 700.052,Z 1046.025,A -85,B 0,C 180,E1 31805.241,E2 31805.241} C_VEL
LIN {X 0,Y 699.157,Z 1066.893,A -85,B 0,C 180,E1 31803.456,E2 31803.456} C_VEL
LIN {X 0,Y 698.395,Z 1086.216,A -85,B 0,C 180,E1 31801.585,E2 31801.585} C_VEL
LIN {X 0,Y 697.757,Z 1103.376,A -85,B 0,C 180,E1 31799.723,E2 31799.723} C_VEL
LIN {X 0,Y 697.193,Z 1120.808,A -85,B 0,C 180,E1 31797.586,E2 31797.586} C_VEL
LIN {X 0,Y 696.762,Z 1135.049,A -85,B 0,C 180,E1 31795.59,E2 31795.59} C_VEL
LIN {X 0,Y 696.455,Z 1147.553,A -85,B 0,C 180,E1 31793.612,E2 31793.612} C_VEL
LIN {X 0,Y 696.233,Z 1159.598,A -85,B 0,C 180,E1 31791.393,E2 31791.393} C_VEL
LIN {X 0,Y 696.072,Z 1168.887,A -85,B 0,C 180,E1 31789.379,E2 31789.379} C_VEL
LIN {X 0,Y 695.999,Z 1176.438,A -85,B 0,C 180,E1 31787.46,E2 31787.46} C_VEL
LIN {X 0,Y 695.947,Z 1183.257,A -85,B 0,C 180,E1 31785.328,E2 31785.328} C_VEL
LIN {X 0,Y 695.918,Z 1188.639,A -85,B 0,C 180,E1 31783.121,E2 31783.121} C_VEL
LIN {X 0,Y 695.911,Z 1192.232,A -85,B 0,C 180,E1 31781.016,E2 31781.016} C_VEL
LIN {X 0,Y 695.908,Z 1194.384,A -85,B 0,C 180,E1 31778.843,E2 31778.843} C_VEL
LIN {X 0,Y 695.904,Z 1194.889,A -85,B 0,C 180,E1 31776.517,E2 31776.517} C_VEL
LIN {X 0,Y 695.907,Z 1193.935,A -85,B 0,C 180,E1 31774.45,E2 31774.45} C_VEL
LIN {X 0,Y 695.916,Z 1191.255,A -85,B 0,C 180,E1 31772.223,E2 31772.223} C_VEL
LIN {X 0,Y 695.933,Z 1187.089,A -85,B 0,C 180,E1 31770.082,E2 31770.082} C_VEL
LIN {X 0,Y 695.967,Z 1181.376,A -85,B 0,C 180,E1 31767.942,E2 31767.942} C_VEL
LIN {X 0,Y 696.043,Z 1173.746,A -85,B 0,C 180,E1 31765.716,E2 31765.716} C_VEL
LIN {X 0,Y 696.152,Z 1163.891,A -85,B 0,C 180,E1 31763.402,E2 31763.402} C_VEL
LIN {X 0,Y 696.346,Z 1153.794,A -85,B 0,C 180,E1 31761.412,E2 31761.412} C_VEL
LIN {X 0,Y 696.61,Z 1142.157,A -85,B 0,C 180,E1 31759.413,E2 31759.413} C_VEL
LIN {X 0,Y 697.002,Z 1126.951,A -85,B 0,C 180,E1 31757.153,E2 31757.153} C_VEL
LIN {X 0,Y 697.452,Z 1112.026,A -85,B 0,C 180,E1 31755.216,E2 31755.216} C_VEL
LIN {X 0,Y 698.034,Z 1095.186,A -85,B 0,C 180,E1 31753.267,E2 31753.267} C_VEL
LIN {X 0,Y 698.761,Z 1076.83,A -85,B 0,C 180,E1 31751.392,E2 31751.392} C_VEL
LIN {X 0,Y 699.548,Z 1057.122,A -85,B 0,C 180,E1 31749.589,E2 31749.589} C_VEL
LIN {X 0,Y 700.499,Z 1035.747,A -85,B 0,C 180,E1 31747.863,E2 31747.863} C_VEL
LIN {X 0,Y 701.506,Z 1013.4,A -85,B 0,C 180,E1 31746.256,E2 31746.256} C_VEL
LIN {X 0,Y 702.571,Z 989.134,A -85,B 0,C 180,E1 31744.726,E2 31744.726} C_VEL
LIN {X 0,Y 703.599,Z 966.086,A -85,B 0,C 180,E1 31743.454,E2 31743.454} C_VEL
LIN {X 0,Y 704.566,Z 943.355,A -85,B 0,C 180,E1 31742.351,E2 31742.351} C_VEL
LIN {X 0,Y 705.564,Z 916.725,A -85,B 0,C 180,E1 31741.242,E2 31741.242} C_VEL
LIN {X 0,Y 706.449,Z 891.715,A -85,B 0,C 180,E1 31740.371,E2 31740.371} C_VEL
LIN {X 0,Y 707.232,Z 866.756,A -85,B 0,C 180,E1 31739.653,E2 31739.653} C_VEL
LIN {X 0,Y 707.951,Z 839.57,A -85,B 0,C 180,E1 31739.037,E2 31739.037} C_VEL
LIN {X 0,Y 708.428,Z 813.636,A -85,B 0,C 180,E1 31738.608,E2 31738.608} C_VEL
LIN {X 0,Y 710.3,Z 589.985,A -85,B 0,C 180,E1 31735.837,E2 31735.837} C_VEL
LIN {X 0,Y 712.154,Z 378.405,A -85,B 0,C 180,E1 31733.136,E2 31733.136} C_VEL
LIN {X 0,Y 712.175,Z 358.145,A -85,B 0,C 180,E1 31732.86,E2 31732.86} C_VEL
LIN {X 0,Y 710.77,Z 353.755,A -85,B 0,C 180,E1 31732.689,E2 31732.689} C_VEL
LIN {X 0,Y 701.997,Z 340.4,A -85,B 0,C 180,E1 31731.77,E2 31731.77} C_VEL
LIN {X 0,Y 697.316,Z 330.501,A -85,B 0,C 180,E1 31730.614,E2 31730.614} C_VEL
LIN {X 0,Y 696.342,Z 327.494,A -85,B 0,C 180,E1 31730.286,E2 31730.286} C_VEL
LIN {X 0,Y 696.314,Z 327.496,A -85,B 0,C 180,E1 31727.219,E2 31727.219} C_VEL
LIN {X 0,Y 696.298,Z 327.494,A -85,B 0,C 180,E1 31724.817,E2 31724.817} C_VEL
LIN {X 0,Y 696.314,Z 327.483,A -85,B 0,C 180,E1 31722.336,E2 31722.336} C_VEL
LIN {X 0,Y 696.349,Z 327.49,A -85,B 0,C 180,E1 31719.289,E2 31719.289} C_VEL
LIN {X 0,Y 696.302,Z 327.49,A -85,B 0,C 180,E1 31716.683,E2 31716.683} C_VEL
LIN {X 0,Y 696.307,Z 327.487,A -85,B 0,C 180,E1 31714.257,E2 31714.257} C_VEL
LIN {X 0,Y 696.391,Z 327.488,A -85,B 0,C 180,E1 31711.317,E2 31711.317} C_VEL
LIN {X 0,Y 696.306,Z 327.476,A -85,B 0,C 180,E1 31708.567,E2 31708.567} C_VEL
LIN {X 0,Y 696.306,Z 327.484,A -85,B 0,C 180,E1 31706.158,E2 31706.158} C_VEL
LIN {X 0,Y 696.371,Z 327.485,A -85,B 0,C 180,E1 31703.437,E2 31703.437} C_VEL
LIN {X 0,Y 696.32,Z 327.482,A -85,B 0,C 180,E1 31700.51,E2 31700.51} C_VEL
LIN {X 0,Y 696.306,Z 327.489,A -85,B 0,C 180,E1 31698.07,E2 31698.07} C_VEL
LIN {X 0,Y 696.326,Z 327.488,A -85,B 0,C 180,E1 31695.576,E2 31695.576} C_VEL
LIN {X 0,Y 696.337,Z 327.488,A -85,B 0,C 180,E1 31692.438,E2 31692.438} C_VEL
LIN {X 0,Y 696.308,Z 327.484,A -85,B 0,C 180,E1 31689.919,E2 31689.919} C_VEL
LIN {X 0,Y 696.318,Z 327.489,A -85,B 0,C 180,E1 31687.509,E2 31687.509} C_VEL
LIN {X 0,Y 696.385,Z 327.486,A -85,B 0,C 180,E1 31684.529,E2 31684.529} C_VEL
LIN {X 0,Y 696.313,Z 327.487,A -85,B 0,C 180,E1 31681.81,E2 31681.81} C_VEL
LIN {X 0,Y 696.312,Z 327.487,A -85,B 0,C 180,E1 31679.424,E2 31679.424} C_VEL
LIN {X 0,Y 696.392,Z 327.488,A -85,B 0,C 180,E1 31676.625,E2 31676.625} C_VEL
LIN {X 0,Y 696.324,Z 327.487,A -85,B 0,C 180,E1 31673.735,E2 31673.735} C_VEL
LIN {X 0,Y 696.314,Z 327.486,A -85,B 0,C 180,E1 31671.245,E2 31671.245} C_VEL
LIN {X 0,Y 696.381,Z 327.478,A -85,B 0,C 180,E1 31668.487,E2 31668.487} C_VEL
LIN {X 0,Y 696.325,Z 327.483,A -85,B 0,C 180,E1 31665.531,E2 31665.531} C_VEL
LIN {X 0,Y 696.316,Z 327.488,A -85,B 0,C 180,E1 31663.052,E2 31663.052} C_VEL
LIN {X 0,Y 696.382,Z 327.469,A -85,B 0,C 180,E1 31660.28,E2 31660.28} C_VEL
LIN {X 0,Y 696.332,Z 327.485,A -85,B 0,C 180,E1 31657.367,E2 31657.367} C_VEL
LIN {X 0,Y 696.316,Z 327.47,A -85,B 0,C 180,E1 31654.846,E2 31654.846} C_VEL
LIN {X 0,Y 696.382,Z 327.489,A -85,B 0,C 180,E1 31652.09,E2 31652.09} C_VEL
LIN {X 0,Y 696.337,Z 327.484,A -85,B 0,C 180,E1 31649.161,E2 31649.161} C_VEL
LIN {X 0,Y 696.32,Z 327.485,A -85,B 0,C 180,E1 31646.635,E2 31646.635} C_VEL
LIN {X 0,Y 696.388,Z 327.489,A -85,B 0,C 180,E1 31643.834,E2 31643.834} C_VEL
LIN {X 0,Y 696.331,Z 327.494,A -85,B 0,C 180,E1 31640.84,E2 31640.84} C_VEL
LIN {X 0,Y 696.322,Z 327.49,A -85,B 0,C 180,E1 31638.427,E2 31638.427} C_VEL
LIN {X 0,Y 696.408,Z 327.533,A -85,B 0,C 180,E1 31637.398,E2 31637.398} C_VEL
LIN {X 0,Y 697.789,Z 331.159,A -85,B 0,C 180,E1 31636.993,E2 31636.993} C_VEL
LIN {X 0,Y 704.479,Z 345.708,A -85,B 0,C 180,E1 31635.321,E2 31635.321} C_VEL
LIN {X 0,Y 707.094,Z 351.223,A -85,B 0,C 180,E1 31634.732,E2 31634.732} C_VEL
LIN {X 0,Y 708.616,Z 354.193,A -85,B 0,C 180,E1 31634.569,E2 31634.569} C_VEL
LIN {X 0,Y 712.334,Z 368.711,A -85,B 0,C 180,E1 31634.075,E2 31634.075} C_VEL
LIN {X 0,Y 710.469,Z 580.092,A -85,B 0,C 180,E1 31631.368,E2 31631.368} C_VEL
LIN {X 0,Y 708.649,Z 803.484,A -85,B 0,C 180,E1 31628.601,E2 31628.601} C_VEL
LIN {X 0,Y 708.214,Z 836.816,A -85,B 0,C 180,E1 31628.148,E2 31628.148} C_VEL
LIN {X 0,Y 707.575,Z 863.584,A -85,B 0,C 180,E1 31627.622,E2 31627.622} C_VEL
LIN {X 0,Y 706.893,Z 888.794,A -85,B 0,C 180,E1 31626.977,E2 31626.977} C_VEL
LIN {X 0,Y 705.97,Z 916.909,A -85,B 0,C 180,E1 31626.071,E2 31626.071} C_VEL
LIN {X 0,Y 705.111,Z 939.393,A -85,B 0,C 180,E1 31625.204,E2 31625.204} C_VEL
LIN {X 0,Y 704.278,Z 959.721,A -85,B 0,C 180,E1 31624.306,E2 31624.306} C_VEL
LIN {X 0,Y 703.406,Z 979.97,A -85,B 0,C 180,E1 31623.296,E2 31623.296} C_VEL
LIN {X 0,Y 702.349,Z 1004.214,A -85,B 0,C 180,E1 31621.929,E2 31621.929} C_VEL
LIN {X 0,Y 701.36,Z 1026.257,A -85,B 0,C 180,E1 31620.498,E2 31620.498} C_VEL
LIN {X 0,Y 700.54,Z 1044.723,A -85,B 0,C 180,E1 31619.166,E2 31619.166} C_VEL
LIN {X 0,Y 699.646,Z 1065.15,A -85,B 0,C 180,E1 31617.536,E2 31617.536} C_VEL
LIN {X 0,Y 698.843,Z 1084.524,A -85,B 0,C 180,E1 31615.782,E2 31615.782} C_VEL
LIN {X 0,Y 698.206,Z 1100.547,A -85,B 0,C 180,E1 31614.177,E2 31614.177} C_VEL
LIN {X 0,Y 697.593,Z 1118.362,A -85,B 0,C 180,E1 31612.189,E2 31612.189} C_VEL
LIN {X 0,Y 697.09,Z 1133.813,A -85,B 0,C 180,E1 31610.223,E2 31610.223} C_VEL
LIN {X 0,Y 696.733,Z 1146.592,A -85,B 0,C 180,E1 31608.404,E2 31608.404} C_VEL
LIN {X 0,Y 696.411,Z 1159.879,A -85,B 0,C 180,E1 31606.258,E2 31606.258} C_VEL
LIN {X 0,Y 696.216,Z 1170.714,A -85,B 0,C 180,E1 31604.205,E2 31604.205} C_VEL
LIN {X 0,Y 696.087,Z 1178.793,A -85,B 0,C 180,E1 31602.442,E2 31602.442} C_VEL
LIN {X 0,Y 695.998,Z 1186.427,A -85,B 0,C 180,E1 31600.512,E2 31600.512} C_VEL
LIN {X 0,Y 695.949,Z 1193.595,A -85,B 0,C 180,E1 31598.26,E2 31598.26} C_VEL
LIN {X 0,Y 695.92,Z 1198.937,A -85,B 0,C 180,E1 31596.02,E2 31596.02} C_VEL
LIN {X 0,Y 695.908,Z 1202.484,A -85,B 0,C 180,E1 31593.872,E2 31593.872} C_VEL
LIN {X 0,Y 695.908,Z 1204.549,A -85,B 0,C 180,E1 31591.647,E2 31591.647} C_VEL
LIN {X 0,Y 695.89,Z 1204.872,A -85,B 0,C 180,E1 31589.506,E2 31589.506} C_VEL
LIN {X 0,Y 695.907,Z 1203.961,A -85,B 0,C 180,E1 31587.53,E2 31587.53} C_VEL
LIN {X 0,Y 695.909,Z 1201.428,A -85,B 0,C 180,E1 31585.385,E2 31585.385} C_VEL
LIN {X 0,Y 695.922,Z 1197.348,A -85,B 0,C 180,E1 31583.234,E2 31583.234} C_VEL
LIN {X 0,Y 695.957,Z 1191.391,A -85,B 0,C 180,E1 31580.991,E2 31580.991} C_VEL
LIN {X 0,Y 696.017,Z 1184.162,A -85,B 0,C 180,E1 31578.871,E2 31578.871} C_VEL
LIN {X 0,Y 696.165,Z 1173.94,A -85,B 0,C 180,E1 31576.461,E2 31576.461} C_VEL
LIN {X 0,Y 696.309,Z 1164.535,A -85,B 0,C 180,E1 31574.595,E2 31574.595} C_VEL
LIN {X 0,Y 696.535,Z 1154.749,A -85,B 0,C 180,E1 31572.886,E2 31572.886} C_VEL
LIN {X 0,Y 696.81,Z 1143.682,A -85,B 0,C 180,E1 31571.164,E2 31571.164} C_VEL
LIN {X 0,Y 697.256,Z 1128.618,A -85,B 0,C 180,E1 31569.08,E2 31569.08} C_VEL
LIN {X 0,Y 697.77,Z 1112.484,A -85,B 0,C 180,E1 31567.133,E2 31567.133} C_VEL
LIN {X 0,Y 698.354,Z 1097.132,A -85,B 0,C 180,E1 31565.468,E2 31565.468} C_VEL
LIN {X 0,Y 699.102,Z 1077.878,A -85,B 0,C 180,E1 31563.59,E2 31563.59} C_VEL
LIN {X 0,Y 699.908,Z 1059.06,A -85,B 0,C 180,E1 31561.966,E2 31561.966} C_VEL
LIN {X 0,Y 700.676,Z 1041.637,A -85,B 0,C 180,E1 31560.601,E2 31560.601} C_VEL
LIN {X 0,Y 701.655,Z 1019.543,A -85,B 0,C 180,E1 31559.041,E2 31559.041} C_VEL
LIN {X 0,Y 702.662,Z 997.051,A -85,B 0,C 180,E1 31557.654,E2 31557.654} C_VEL
LIN {X 0,Y 703.513,Z 977.658,A -85,B 0,C 180,E1 31556.583,E2 31556.583} C_VEL
LIN {X 0,Y 704.372,Z 957.732,A -85,B 0,C 180,E1 31555.6,E2 31555.6} C_VEL
LIN {X 0,Y 705.354,Z 933.855,A -85,B 0,C 180,E1 31554.566,E2 31554.566} C_VEL
LIN {X 0,Y 706.253,Z 907.072,A -85,B 0,C 180,E1 31553.591,E2 31553.591} C_VEL
LIN {X 0,Y 707.026,Z 883.676,A -85,B 0,C 180,E1 31552.881,E2 31552.881} C_VEL
LIN {X 0,Y 707.751,Z 857.861,A -85,B 0,C 180,E1 31552.252,E2 31552.252} C_VEL
LIN {X 0,Y 708.321,Z 830.109,A -85,B 0,C 180,E1 31551.745,E2 31551.745} C_VEL
LIN {X 0,Y 709.321,Z 718.522,A -85,B 0,C 180,E1 31550.357,E2 31550.357} C_VEL
LIN {X 0,Y 711.17,Z 499.459,A -85,B 0,C 180,E1 31547.61,E2 31547.61} C_VEL
LIN {X 0,Y 712.169,Z 367.486,A -85,B 0,C 180,E1 31545.895,E2 31545.895} C_VEL
LIN {X 0,Y 708.03,Z 352.733,A -85,B 0,C 180,E1 31545.364,E2 31545.364} C_VEL
LIN {X 0,Y 706.447,Z 350.084,A -85,B 0,C 180,E1 31545.162,E2 31545.162} C_VEL
LIN {X 0,Y 699.859,Z 335.524,A -85,B 0,C 180,E1 31543.522,E2 31543.522} C_VEL
LIN {X 0,Y 696.503,Z 328.119,A -85,B 0,C 180,E1 31542.656,E2 31542.656} C_VEL
LIN {X 0,Y 696.404,Z 327.488,A -85,B 0,C 180,E1 31542.563,E2 31542.563} C_VEL
LIN {X 0,Y 696.332,Z 327.494,A -85,B 0,C 180,E1 31539.679,E2 31539.679} C_VEL
LIN {X 0,Y 696.331,Z 327.489,A -85,B 0,C 180,E1 31537.163,E2 31537.163} C_VEL
LIN {X 0,Y 696.407,Z 327.484,A -85,B 0,C 180,E1 31534.21,E2 31534.21} C_VEL
LIN {X 0,Y 696.329,Z 327.475,A -85,B 0,C 180,E1 31531.311,E2 31531.311} C_VEL
LIN {X 0,Y 696.343,Z 327.486,A -85,B 0,C 180,E1 31528.753,E2 31528.753} C_VEL
LIN {X 0,Y 696.376,Z 327.485,A -85,B 0,C 180,E1 31525.698,E2 31525.698} C_VEL
LIN {X 0,Y 696.329,Z 327.476,A -85,B 0,C 180,E1 31522.991,E2 31522.991} C_VEL
LIN {X 0,Y 696.364,Z 327.482,A -85,B 0,C 180,E1 31520.333,E2 31520.333} C_VEL
LIN {X 0,Y 696.348,Z 327.478,A -85,B 0,C 180,E1 31517.205,E2 31517.205} C_VEL
LIN {X 0,Y 696.336,Z 327.486,A -85,B 0,C 180,E1 31514.554,E2 31514.554} C_VEL
LIN {X 0,Y 696.405,Z 327.468,A -85,B 0,C 180,E1 31511.68,E2 31511.68} C_VEL
LIN {X 0,Y 696.337,Z 327.485,A -85,B 0,C 180,E1 31508.755,E2 31508.755} C_VEL
LIN {X 0,Y 696.341,Z 327.472,A -85,B 0,C 180,E1 31506.182,E2 31506.182} C_VEL
LIN {X 0,Y 696.4,Z 327.484,A -85,B 0,C 180,E1 31503.21,E2 31503.21} C_VEL
LIN {X 0,Y 696.335,Z 327.481,A -85,B 0,C 180,E1 31500.411,E2 31500.411} C_VEL
LIN {X 0,Y 696.368,Z 327.483,A -85,B 0,C 180,E1 31497.696,E2 31497.696} C_VEL
LIN {X 0,Y 696.356,Z 327.487,A -85,B 0,C 180,E1 31494.562,E2 31494.562} C_VEL
LIN {X 0,Y 696.338,Z 327.482,A -85,B 0,C 180,E1 31491.91,E2 31491.91} C_VEL
LIN {X 0,Y 696.403,Z 327.475,A -85,B 0,C 180,E1 31488.991,E2 31488.991} C_VEL
LIN {X 0,Y 696.34,Z 327.474,A -85,B 0,C 180,E1 31486.084,E2 31486.084} C_VEL
LIN {X 0,Y 696.359,Z 327.482,A -85,B 0,C 180,E1 31483.397,E2 31483.397} C_VEL
LIN {X 0,Y 696.373,Z 327.477,A -85,B 0,C 180,E1 31480.28,E2 31480.28} C_VEL
LIN {X 0,Y 696.341,Z 327.483,A -85,B 0,C 180,E1 31477.545,E2 31477.545} C_VEL
LIN {X 0,Y 696.357,Z 327.48,A -85,B 0,C 180,E1 31475.166,E2 31475.166} C_VEL
LIN {X 0,Y 695.416,Z 327.606,A -85,B 0,C 180,E1 31474.532,E2 31474.532} C_VEL
LIN {X 0,Y 689.018,Z 328.405,A -85,B 0,C 180,E1 31472.757,E2 31472.757} C_VEL
LIN {X 0,Y 688.463,Z 328.477,A -85,B 0,C 180,E1 31472.295,E2 31472.295} C_VEL
LIN {X 0,Y 688.405,Z 328.474,A -85,B 0,C 180,E1 31469.445,E2 31469.445} C_VEL
LIN {X 0,Y 688.458,Z 328.475,A -85,B 0,C 180,E1 31466.602,E2 31466.602} C_VEL
LIN {X 0,Y 688.478,Z 328.572,A -85,B 0,C 180,E1 31464.228,E2 31464.228} C_VEL
LIN {X 0,Y 689.75,Z 331.962,A -85,B 0,C 180,E1 31463.842,E2 31463.842} C_VEL
LIN {X 0,Y 694.211,Z 341.284,A -85,B 0,C 180,E1 31462.75,E2 31462.75} C_VEL
LIN {X 0,Y 706.2,Z 359.424,A -85,B 0,C 180,E1 31461.504,E2 31461.504} C_VEL
LIN {X 0,Y 706.561,Z 362.185,A -85,B 0,C 180,E1 31461.437,E2 31461.437} C_VEL
LIN {X 0,Y 704.449,Z 570.892,A -85,B 0,C 180,E1 31458.745,E2 31458.745} C_VEL
LIN {X 0,Y 702.381,Z 794.573,A -85,B 0,C 180,E1 31455.951,E2 31455.951} C_VEL
LIN {X 0,Y 701.884,Z 827.22,A -85,B 0,C 180,E1 31455.501,E2 31455.501} C_VEL
LIN {X 0,Y 701.208,Z 852.919,A -85,B 0,C 180,E1 31454.994,E2 31454.994} C_VEL
LIN {X 0,Y 700.423,Z 878.82,A -85,B 0,C 180,E1 31454.331,E2 31454.331} C_VEL
LIN {X 0,Y 699.427,Z 905.565,A -85,B 0,C 180,E1 31453.469,E2 31453.469} C_VEL
LIN {X 0,Y 698.44,Z 929.087,A -85,B 0,C 180,E1 31452.564,E2 31452.564} C_VEL
LIN {X 0,Y 697.35,Z 952.476,A -85,B 0,C 180,E1 31451.516,E2 31451.516} C_VEL
LIN {X 0,Y 696.146,Z 976.71,A -85,B 0,C 180,E1 31450.265,E2 31450.265} C_VEL
LIN {X 0,Y 695.006,Z 999.838,A -85,B 0,C 180,E1 31448.892,E2 31448.892} C_VEL
LIN {X 0,Y 693.83,Z 1022.787,A -85,B 0,C 180,E1 31447.35,E2 31447.35} C_VEL
LIN {X 0,Y 692.652,Z 1046.007,A -85,B 0,C 180,E1 31445.573,E2 31445.573} C_VEL
LIN {X 0,Y 691.668,Z 1066.808,A -85,B 0,C 180,E1 31443.774,E2 31443.774} C_VEL
LIN {X 0,Y 690.743,Z 1086.759,A -85,B 0,C 180,E1 31441.819,E2 31441.819} C_VEL
LIN {X 0,Y 689.984,Z 1105.019,A -85,B 0,C 180,E1 31439.804,E2 31439.804} C_VEL
LIN {X 0,Y 689.341,Z 1122.094,A -85,B 0,C 180,E1 31437.655,E2 31437.655} C_VEL
LIN {X 0,Y 688.865,Z 1136.27,A -85,B 0,C 180,E1 31435.628,E2 31435.628} C_VEL
LIN {X 0,Y 688.497,Z 1149.639,A -85,B 0,C 180,E1 31433.448,E2 31433.448} C_VEL
LIN {X 0,Y 688.265,Z 1160.883,A -85,B 0,C 180,E1 31431.296,E2 31431.296} C_VEL
LIN {X 0,Y 688.088,Z 1169.633,A -85,B 0,C 180,E1 31429.348,E2 31429.348} C_VEL
LIN {X 0,Y 688.004,Z 1177.004,A -85,B 0,C 180,E1 31427.42,E2 31427.42} C_VEL
LIN {X 0,Y 687.95,Z 1183.757,A -85,B 0,C 180,E1 31425.252,E2 31425.252} C_VEL
LIN {X 0,Y 687.917,Z 1189.164,A -85,B 0,C 180,E1 31422.934,E2 31422.934} C_VEL
LIN {X 0,Y 687.909,Z 1192.56,A -85,B 0,C 180,E1 31420.807,E2 31420.807} C_VEL
LIN {X 0,Y 687.908,Z 1194.555,A -85,B 0,C 180,E1 31418.61,E2 31418.61} C_VEL
LIN {X 0,Y 687.906,Z 1194.865,A -85,B 0,C 180,E1 31416.426,E2 31416.426} C_VEL
LIN {X 0,Y 687.907,Z 1193.931,A -85,B 0,C 180,E1 31414.418,E2 31414.418} C_VEL
LIN {X 0,Y 687.918,Z 1191.252,A -85,B 0,C 180,E1 31412.166,E2 31412.166} C_VEL
LIN {X 0,Y 687.94,Z 1187.083,A -85,B 0,C 180,E1 31410,E2 31410} C_VEL
LIN {X 0,Y 687.976,Z 1181.369,A -85,B 0,C 180,E1 31407.834,E2 31407.834} C_VEL
LIN {X 0,Y 688.063,Z 1173.742,A -85,B 0,C 180,E1 31405.583,E2 31405.583} C_VEL
LIN {X 0,Y 688.187,Z 1163.891,A -85,B 0,C 180,E1 31403.242,E2 31403.242} C_VEL
LIN {X 0,Y 688.414,Z 1153.796,A -85,B 0,C 180,E1 31401.228,E2 31401.228} C_VEL
LIN {X 0,Y 688.725,Z 1141.655,A -85,B 0,C 180,E1 31399.122,E2 31399.122} C_VEL
LIN {X 0,Y 689.186,Z 1126.337,A -85,B 0,C 180,E1 31396.834,E2 31396.834} C_VEL
LIN {X 0,Y 689.761,Z 1110.668,A -85,B 0,C 180,E1 31394.789,E2 31394.789} C_VEL
LIN {X 0,Y 690.484,Z 1092.843,A -85,B 0,C 180,E1 31392.732,E2 31392.732} C_VEL
LIN {X 0,Y 691.328,Z 1073.29,A -85,B 0,C 180,E1 31390.746,E2 31390.746} C_VEL
LIN {X 0,Y 692.371,Z 1052.04,A -85,B 0,C 180,E1 31388.837,E2 31388.837} C_VEL
LIN {X 0,Y 693.488,Z 1029.456,A -85,B 0,C 180,E1 31387.045,E2 31387.045} C_VEL
LIN {X 0,Y 694.725,Z 1005.443,A -85,B 0,C 180,E1 31385.377,E2 31385.377} C_VEL
LIN {X 0,Y 695.926,Z 981.574,A -85,B 0,C 180,E1 31383.919,E2 31383.919} C_VEL
LIN {X 0,Y 697.193,Z 955.632,A -85,B 0,C 180,E1 31382.544,E2 31382.544} C_VEL
LIN {X 0,Y 698.34,Z 931.107,A -85,B 0,C 180,E1 31381.432,E2 31381.432} C_VEL
LIN {X 0,Y 699.319,Z 908.286,A -85,B 0,C 180,E1 31380.539,E2 31380.539} C_VEL
LIN {X 0,Y 700.327,Z 881.603,A -85,B 0,C 180,E1 31379.66,E2 31379.66} C_VEL
LIN {X 0,Y 701.179,Z 854.233,A -85,B 0,C 180,E1 31378.945,E2 31378.945} C_VEL
LIN {X 0,Y 701.833,Z 829.115,A -85,B 0,C 180,E1 31378.442,E2 31378.442} C_VEL
LIN {X 0,Y 702.332,Z 799.854,A -85,B 0,C 180,E1 31378.024,E2 31378.024} C_VEL
LIN {X 0,Y 704.373,Z 578.749,A -85,B 0,C 180,E1 31375.264,E2 31375.264} C_VEL
LIN {X 0,Y 706.511,Z 366.36,A -85,B 0,C 180,E1 31372.527,E2 31372.527} C_VEL
LIN {X 0,Y 706.399,Z 360.436,A -85,B 0,C 180,E1 31372.436,E2 31372.436} C_VEL
LIN {X 0,Y 705.41,Z 358.083,A -85,B 0,C 180,E1 31372.324,E2 31372.324} C_VEL
LIN {X 0,Y 693.785,Z 340.63,A -85,B 0,C 180,E1 31371.101,E2 31371.101} C_VEL
LIN {X 0,Y 688.574,Z 329.267,A -85,B 0,C 180,E1 31369.747,E2 31369.747} C_VEL
LIN {X 0,Y 688.42,Z 328.478,A -85,B 0,C 180,E1 31369.654,E2 31369.654} C_VEL
LIN {X 0,Y 688.362,Z 328.486,A -85,B 0,C 180,E1 31366.94,E2 31366.94} C_VEL
LIN {X 0,Y 688.369,Z 328.484,A -85,B 0,C 180,E1 31364.506,E2 31364.506} C_VEL
LIN {X 0,Y 688.447,Z 328.465,A -85,B 0,C 180,E1 31361.586,E2 31361.586} C_VEL
LIN {X 0,Y 688.365,Z 328.48,A -85,B 0,C 180,E1 31358.76,E2 31358.76} C_VEL
LIN {X 0,Y 688.367,Z 328.479,A -85,B 0,C 180,E1 31356.345,E2 31356.345} C_VEL
LIN {X 0,Y 688.458,Z 328.478,A -85,B 0,C 180,E1 31353.498,E2 31353.498} C_VEL
LIN {X 0,Y 688.372,Z 328.479,A -85,B 0,C 180,E1 31350.654,E2 31350.654} C_VEL
LIN {X 0,Y 688.365,Z 328.464,A -85,B 0,C 180,E1 31348.264,E2 31348.264} C_VEL
LIN {X 0,Y 688.42,Z 328.474,A -85,B 0,C 180,E1 31345.555,E2 31345.555} C_VEL
LIN {X 0,Y 688.378,Z 328.462,A -85,B 0,C 180,E1 31342.515,E2 31342.515} C_VEL
LIN {X 0,Y 688.366,Z 328.471,A -85,B 0,C 180,E1 31340.048,E2 31340.048} C_VEL
LIN {X 0,Y 688.415,Z 328.479,A -85,B 0,C 180,E1 31337.403,E2 31337.403} C_VEL
LIN {X 0,Y 688.385,Z 328.475,A -85,B 0,C 180,E1 31334.351,E2 31334.351} C_VEL
LIN {X 0,Y 688.368,Z 328.478,A -85,B 0,C 180,E1 31331.903,E2 31331.903} C_VEL
LIN {X 0,Y 688.394,Z 328.474,A -85,B 0,C 180,E1 31329.363,E2 31329.363} C_VEL
LIN {X 0,Y 688.397,Z 328.472,A -85,B 0,C 180,E1 31326.254,E2 31326.254} C_VEL
LIN {X 0,Y 688.372,Z 328.477,A -85,B 0,C 180,E1 31323.748,E2 31323.748} C_VEL
LIN {X 0,Y 688.394,Z 328.477,A -85,B 0,C 180,E1 31321.165,E2 31321.165} C_VEL
LIN {X 0,Y 688.397,Z 328.476,A -85,B 0,C 180,E1 31318.002,E2 31318.002} C_VEL
LIN {X 0,Y 688.372,Z 328.471,A -85,B 0,C 180,E1 31315.501,E2 31315.501} C_VEL
LIN {X 0,Y 688.393,Z 328.479,A -85,B 0,C 180,E1 31312.992,E2 31312.992} C_VEL
LIN {X 0,Y 688.409,Z 328.474,A -85,B 0,C 180,E1 31309.878,E2 31309.878} C_VEL
LIN {X 0,Y 688.373,Z 328.457,A -85,B 0,C 180,E1 31307.245,E2 31307.245} C_VEL
LIN {X 0,Y 688.404,Z 328.475,A -85,B 0,C 180,E1 31304.668,E2 31304.668} C_VEL
LIN {X 0,Y 688.394,Z 328.458,A -85,B 0,C 180,E1 31301.522,E2 31301.522} C_VEL
LIN {X 0,Y 688.377,Z 328.474,A -85,B 0,C 180,E1 31298.975,E2 31298.975} C_VEL
LIN {X 0,Y 688.414,Z 328.471,A -85,B 0,C 180,E1 31296.367,E2 31296.367} C_VEL
LIN {X 0,Y 688.397,Z 328.476,A -85,B 0,C 180,E1 31293.284,E2 31293.284} C_VEL
LIN {X 0,Y 688.38,Z 328.476,A -85,B 0,C 180,E1 31290.787,E2 31290.787} C_VEL
LIN {X 0,Y 688.415,Z 328.477,A -85,B 0,C 180,E1 31288.174,E2 31288.174} C_VEL
LIN {X 0,Y 688.401,Z 328.478,A -85,B 0,C 180,E1 31285.091,E2 31285.091} C_VEL
LIN {X 0,Y 688.384,Z 328.481,A -85,B 0,C 180,E1 31282.471,E2 31282.471} C_VEL
LIN {X 0,Y 688.465,Z 328.477,A -85,B 0,C 180,E1 31279.628,E2 31279.628} C_VEL
LIN {X 0,Y 688.42,Z 328.592,A -85,B 0,C 180,E1 31278.041,E2 31278.041} C_VEL
LIN {X 0,Y 689.876,Z 332.124,A -85,B 0,C 180,E1 31277.626,E2 31277.626} C_VEL
LIN {X 0,Y 698.082,Z 349.884,A -85,B 0,C 180,E1 31275.539,E2 31275.539} C_VEL
LIN {X 0,Y 699.256,Z 351.997,A -85,B 0,C 180,E1 31275.361,E2 31275.361} C_VEL
LIN {X 0,Y 703.374,Z 358.355,A -85,B 0,C 180,E1 31274.932,E2 31274.932} C_VEL
LIN {X 0,Y 706.551,Z 371.029,A -85,B 0,C 180,E1 31274.499,E2 31274.499} C_VEL
LIN {X 0,Y 704.431,Z 582.815,A -85,B 0,C 180,E1 31271.766,E2 31271.766} C_VEL
LIN {X 0,Y 702.367,Z 806,A -85,B 0,C 180,E1 31268.978,E2 31268.978} C_VEL
LIN {X 0,Y 701.865,Z 838.3,A -85,B 0,C 180,E1 31268.528,E2 31268.528} C_VEL
LIN {X 0,Y 701.168,Z 864.281,A -85,B 0,C 180,E1 31268.009,E2 31268.009} C_VEL
LIN {X 0,Y 700.391,Z 889.517,A -85,B 0,C 180,E1 31267.356,E2 31267.356} C_VEL
LIN {X 0,Y 699.346,Z 917.484,A -85,B 0,C 180,E1 31266.444,E2 31266.444} C_VEL
LIN {X 0,Y 698.408,Z 939.439,A -85,B 0,C 180,E1 31265.591,E2 31265.591} C_VEL
LIN {X 0,Y 697.472,Z 959.724,A -85,B 0,C 180,E1 31264.689,E2 31264.689} C_VEL
LIN {X 0,Y 696.515,Z 979.444,A -85,B 0,C 180,E1 31263.699,E2 31263.699} C_VEL
LIN {X 0,Y 695.398,Z 1001.889,A -85,B 0,C 180,E1 31262.432,E2 31262.432} C_VEL
LIN {X 0,Y 694.216,Z 1024.924,A -85,B 0,C 180,E1 31260.942,E2 31260.942} C_VEL
LIN {X 0,Y 693.268,Z 1043.78,A -85,B 0,C 180,E1 31259.576,E2 31259.576} C_VEL
LIN {X 0,Y 692.351,Z 1062.382,A -85,B 0,C 180,E1 31258.086,E2 31258.086} C_VEL
LIN {X 0,Y 691.305,Z 1083.593,A -85,B 0,C 180,E1 31256.176,E2 31256.176} C_VEL
LIN {X 0,Y 690.611,Z 1099.695,A -85,B 0,C 180,E1 31254.552,E2 31254.552} C_VEL
LIN {X 0,Y 689.909,Z 1116.495,A -85,B 0,C 180,E1 31252.675,E2 31252.675} C_VEL
LIN {X 0,Y 689.312,Z 1132.526,A -85,B 0,C 180,E1 31250.639,E2 31250.639} C_VEL
LIN {X 0,Y 688.907,Z 1145.025,A -85,B 0,C 180,E1 31248.857,E2 31248.857} C_VEL
LIN {X 0,Y 688.592,Z 1156.316,A -85,B 0,C 180,E1 31247.056,E2 31247.056} C_VEL
LIN {X 0,Y 688.306,Z 1168.607,A -85,B 0,C 180,E1 31244.813,E2 31244.813} C_VEL
LIN {X 0,Y 688.131,Z 1178.079,A -85,B 0,C 180,E1 31242.759,E2 31242.759} C_VEL
LIN {X 0,Y 688.006,Z 1186.016,A -85,B 0,C 180,E1 31240.751,E2 31240.751} C_VEL
LIN {X 0,Y 687.959,Z 1193.11,A -85,B 0,C 180,E1 31238.525,E2 31238.525} C_VEL
LIN {X 0,Y 687.926,Z 1198.594,A -85,B 0,C 180,E1 31236.258,E2 31236.258} C_VEL
LIN {X 0,Y 687.915,Z 1202.263,A -85,B 0,C 180,E1 31234.084,E2 31234.084} C_VEL
LIN {X 0,Y 687.907,Z 1204.438,A -85,B 0,C 180,E1 31231.832,E2 31231.832} C_VEL
LIN {X 0,Y 687.891,Z 1204.894,A -85,B 0,C 180,E1 31229.584,E2 31229.584} C_VEL
LIN {X 0,Y 687.907,Z 1203.959,A -85,B 0,C 180,E1 31227.501,E2 31227.501} C_VEL
LIN {X 0,Y 687.91,Z 1201.428,A -85,B 0,C 180,E1 31225.331,E2 31225.331} C_VEL
LIN {X 0,Y 687.927,Z 1197.152,A -85,B 0,C 180,E1 31223.071,E2 31223.071} C_VEL
LIN {X 0,Y 687.967,Z 1191.388,A -85,B 0,C 180,E1 31220.885,E2 31220.885} C_VEL
LIN {X 0,Y 688.039,Z 1184.277,A -85,B 0,C 180,E1 31218.771,E2 31218.771} C_VEL
LIN {X 0,Y 688.2,Z 1173.939,A -85,B 0,C 180,E1 31216.301,E2 31216.301} C_VEL
LIN {X 0,Y 688.395,Z 1164.291,A -85,B 0,C 180,E1 31214.368,E2 31214.368} C_VEL
LIN {X 0,Y 688.644,Z 1154.228,A -85,B 0,C 180,E1 31212.597,E2 31212.597} C_VEL
LIN {X 0,Y 688.983,Z 1142.519,A -85,B 0,C 180,E1 31210.766,E2 31210.766} C_VEL
LIN {X 0,Y 689.531,Z 1126.514,A -85,B 0,C 180,E1 31208.567,E2 31208.567} C_VEL
LIN {X 0,Y 690.12,Z 1111.233,A -85,B 0,C 180,E1 31206.72,E2 31206.72} C_VEL
LIN {X 0,Y 690.81,Z 1094.573,A -85,B 0,C 180,E1 31204.908,E2 31204.908} C_VEL
LIN {X 0,Y 691.75,Z 1074.836,A -85,B 0,C 180,E1 31203.009,E2 31203.009} C_VEL
LIN {X 0,Y 692.543,Z 1057.953,A -85,B 0,C 180,E1 31201.547,E2 31201.547} C_VEL
LIN {X 0,Y 693.498,Z 1038.972,A -85,B 0,C 180,E1 31200.058,E2 31200.058} C_VEL
LIN {X 0,Y 694.719,Z 1015.179,A -85,B 0,C 180,E1 31198.407,E2 31198.407} C_VEL
LIN {X 0,Y 695.721,Z 995.448,A -85,B 0,C 180,E1 31197.193,E2 31197.193} C_VEL
LIN {X 0,Y 696.697,Z 975.877,A -85,B 0,C 180,E1 31196.113,E2 31196.113} C_VEL
LIN {X 0,Y 697.765,Z 953.709,A -85,B 0,C 180,E1 31195.028,E2 31195.028} C_VEL
LIN {X 0,Y 698.897,Z 927.097,A -85,B 0,C 180,E1 31193.911,E2 31193.911} C_VEL
LIN {X 0,Y 699.79,Z 904.877,A -85,B 0,C 180,E1 31193.123,E2 31193.123} C_VEL
LIN {X 0,Y 700.634,Z 881.957,A -85,B 0,C 180,E1 31192.434,E2 31192.434} C_VEL
LIN {X 0,Y 701.466,Z 854.989,A -85,B 0,C 180,E1 31191.785,E2 31191.785} C_VEL
LIN {X 0,Y 702.071,Z 827.553,A -85,B 0,C 180,E1 31191.303,E2 31191.303} C_VEL
LIN {X 0,Y 704.228,Z 603.934,A -85,B 0,C 180,E1 31188.502,E2 31188.502} C_VEL
LIN {X 0,Y 706.246,Z 399.778,A -85,B 0,C 180,E1 31185.877,E2 31185.877} C_VEL
LIN {X 0,Y 706.388,Z 369.725,A -85,B 0,C 180,E1 31185.47,E2 31185.47} C_VEL
LIN {X 0,Y 702.932,Z 357.343,A -85,B 0,C 180,E1 31185.017,E2 31185.017} C_VEL
LIN {X 0,Y 698.287,Z 350.376,A -85,B 0,C 180,E1 31184.515,E2 31184.515} C_VEL
LIN {X 0,Y 691.524,Z 335.793,A -85,B 0,C 180,E1 31182.811,E2 31182.811} C_VEL
LIN {X 0,Y 689.877,Z 332.121,A -85,B 0,C 180,E1 31182.374,E2 31182.374} C_VEL
LIN {X 0,Y 688.415,Z 328.532,A -85,B 0,C 180,E1 31181.954,E2 31181.954} C_VEL
LIN {X 0,Y 688.387,Z 328.482,A -85,B 0,C 180,E1 31179.402,E2 31179.402} C_VEL
LIN {X 0,Y 688.443,Z 328.476,A -85,B 0,C 180,E1 31176.651,E2 31176.651} C_VEL
LIN {X 0,Y 688.4,Z 328.479,A -85,B 0,C 180,E1 31173.601,E2 31173.601} C_VEL
LIN {X 0,Y 688.393,Z 328.462,A -85,B 0,C 180,E1 31171.025,E2 31171.025} C_VEL
LIN {X 0,Y 688.469,Z 328.467,A -85,B 0,C 180,E1 31168.165,E2 31168.165} C_VEL
LIN {X 0,Y 688.394,Z 328.478,A -85,B 0,C 180,E1 31165.194,E2 31165.194} C_VEL
LIN {X 0,Y 688.4,Z 328.462,A -85,B 0,C 180,E1 31162.638,E2 31162.638} C_VEL
LIN {X 0,Y 688.452,Z 328.475,A -85,B 0,C 180,E1 31159.603,E2 31159.603} C_VEL
LIN {X 0,Y 688.391,Z 328.467,A -85,B 0,C 180,E1 31156.801,E2 31156.801} C_VEL
LIN {X 0,Y 688.43,Z 328.473,A -85,B 0,C 180,E1 31154.123,E2 31154.123} C_VEL
LIN {X 0,Y 688.415,Z 328.474,A -85,B 0,C 180,E1 31151.053,E2 31151.053} C_VEL
LIN {X 0,Y 688.396,Z 328.472,A -85,B 0,C 180,E1 31148.436,E2 31148.436} C_VEL
LIN {X 0,Y 688.465,Z 328.458,A -85,B 0,C 180,E1 31145.584,E2 31145.584} C_VEL
LIN {X 0,Y 688.405,Z 328.468,A -85,B 0,C 180,E1 31142.664,E2 31142.664} C_VEL
LIN {X 0,Y 688.405,Z 328.467,A -85,B 0,C 180,E1 31140,E2 31140} C_VEL
LIN {X 0,Y 688.46,Z 328.464,A -85,B 0,C 180,E1 31137.003,E2 31137.003} C_VEL
LIN {X 0,Y 688.397,Z 328.474,A -85,B 0,C 180,E1 31134.164,E2 31134.164} C_VEL
LIN {X 0,Y 688.433,Z 328.468,A -85,B 0,C 180,E1 31131.48,E2 31131.48} C_VEL
LIN {X 0,Y 688.417,Z 328.478,A -85,B 0,C 180,E1 31128.352,E2 31128.352} C_VEL
LIN {X 0,Y 688.404,Z 328.459,A -85,B 0,C 180,E1 31125.642,E2 31125.642} C_VEL
LIN {X 0,Y 688.467,Z 328.476,A -85,B 0,C 180,E1 31122.679,E2 31122.679} C_VEL
LIN {X 0,Y 688.402,Z 328.472,A -85,B 0,C 180,E1 31119.763,E2 31119.763} C_VEL
LIN {X 0,Y 688.456,Z 328.466,A -85,B 0,C 180,E1 31116.912,E2 31116.912} C_VEL
LIN {X 0,Y 688.414,Z 328.475,A -85,B 0,C 180,E1 31113.843,E2 31113.843} C_VEL
LIN {X 0,Y 688.463,Z 328.477,A -85,B 0,C 180,E1 31112.295,E2 31112.295} C_VEL
LIN {X 0,Y 687.443,Z 328.604,A -85,B 0,C 180,E1 31111.654,E2 31111.654} C_VEL
LIN {X 0,Y 680.997,Z 329.4,A -85,B 0,C 180,E1 31109.858,E2 31109.858} C_VEL
LIN {X 0,Y 680.466,Z 329.463,A -85,B 0,C 180,E1 31109.39,E2 31109.39} C_VEL
LIN {X 0,Y 680.527,Z 329.465,A -85,B 0,C 180,E1 31106.464,E2 31106.464} C_VEL
LIN {X 0,Y 680.493,Z 329.537,A -85,B 0,C 180,E1 31104.882,E2 31104.882} C_VEL
LIN {X 0,Y 681.856,Z 332.98,A -85,B 0,C 180,E1 31104.473,E2 31104.473} C_VEL
LIN {X 0,Y 685.828,Z 341.383,A -85,B 0,C 180,E1 31103.473,E2 31103.473} C_VEL
LIN {X 0,Y 699.087,Z 360.936,A -85,B 0,C 180,E1 31102.059,E2 31102.059} C_VEL
LIN {X 0,Y 700.822,Z 363.911,A -85,B 0,C 180,E1 31101.875,E2 31101.875} C_VEL
LIN {X 0,Y 698.465,Z 571.99,A -85,B 0,C 180,E1 31099.171,E2 31099.171} C_VEL
LIN {X 0,Y 696.146,Z 795.945,A -85,B 0,C 180,E1 31096.35,E2 31096.35} C_VEL
LIN {X 0,Y 695.585,Z 828.034,A -85,B 0,C 180,E1 31095.9,E2 31095.9} C_VEL
LIN {X 0,Y 694.85,Z 853.299,A -85,B 0,C 180,E1 31095.396,E2 31095.396} C_VEL
LIN {X 0,Y 693.957,Z 879.44,A -85,B 0,C 180,E1 31094.721,E2 31094.721} C_VEL
LIN {X 0,Y 692.833,Z 906.303,A -85,B 0,C 180,E1 31093.845,E2 31093.845} C_VEL
LIN {X 0,Y 691.78,Z 928.987,A -85,B 0,C 180,E1 31092.965,E2 31092.965} C_VEL
LIN {X 0,Y 690.534,Z 953.104,A -85,B 0,C 180,E1 31091.875,E2 31091.875} C_VEL
LIN {X 0,Y 689.164,Z 977.598,A -85,B 0,C 180,E1 31090.594,E2 31090.594} C_VEL
LIN {X 0,Y 687.851,Z 1001.201,A -85,B 0,C 180,E1 31089.173,E2 31089.173} C_VEL
LIN {X 0,Y 686.582,Z 1023.459,A -85,B 0,C 180,E1 31087.655,E2 31087.655} C_VEL
LIN {X 0,Y 685.277,Z 1045.99,A -85,B 0,C 180,E1 31085.912,E2 31085.912} C_VEL
LIN {X 0,Y 684.179,Z 1066.902,A -85,B 0,C 180,E1 31084.082,E2 31084.082} C_VEL
LIN {X 0,Y 683.125,Z 1086.684,A -85,B 0,C 180,E1 31082.124,E2 31082.124} C_VEL
LIN {X 0,Y 682.276,Z 1105.011,A -85,B 0,C 180,E1 31080.079,E2 31080.079} C_VEL
LIN {X 0,Y 681.539,Z 1122.091,A -85,B 0,C 180,E1 31077.904,E2 31077.904} C_VEL
LIN {X 0,Y 680.998,Z 1136.389,A -85,B 0,C 180,E1 31075.835,E2 31075.835} C_VEL
LIN {X 0,Y 680.58,Z 1149.635,A -85,B 0,C 180,E1 31073.645,E2 31073.645} C_VEL
LIN {X 0,Y 680.309,Z 1160.888,A -85,B 0,C 180,E1 31071.467,E2 31071.467} C_VEL
LIN {X 0,Y 680.125,Z 1169.641,A -85,B 0,C 180,E1 31069.494,E2 31069.494} C_VEL
LIN {X 0,Y 680.017,Z 1177.309,A -85,B 0,C 180,E1 31067.455,E2 31067.455} C_VEL
LIN {X 0,Y 679.954,Z 1183.95,A -85,B 0,C 180,E1 31065.275,E2 31065.275} C_VEL
LIN {X 0,Y 679.918,Z 1189.166,A -85,B 0,C 180,E1 31063.003,E2 31063.003} C_VEL
LIN {X 0,Y 679.909,Z 1192.563,A -85,B 0,C 180,E1 31060.85,E2 31060.85} C_VEL
LIN {X 0,Y 679.908,Z 1194.556,A -85,B 0,C 180,E1 31058.627,E2 31058.627} C_VEL
LIN {X 0,Y 679.906,Z 1194.865,A -85,B 0,C 180,E1 31056.417,E2 31056.417} C_VEL
LIN {X 0,Y 679.909,Z 1193.916,A -85,B 0,C 180,E1 31054.373,E2 31054.373} C_VEL
LIN {X 0,Y 679.919,Z 1191.249,A -85,B 0,C 180,E1 31052.107,E2 31052.107} C_VEL
LIN {X 0,Y 679.945,Z 1186.883,A -85,B 0,C 180,E1 31049.832,E2 31049.832} C_VEL
LIN {X 0,Y 679.989,Z 1181.117,A -85,B 0,C 180,E1 31047.64,E2 31047.64} C_VEL
LIN {X 0,Y 680.077,Z 1173.112,A -85,B 0,C 180,E1 31045.277,E2 31045.277} C_VEL
LIN {X 0,Y 680.24,Z 1163.489,A -85,B 0,C 180,E1 31042.993,E2 31042.993} C_VEL
LIN {X 0,Y 680.484,Z 1153.345,A -85,B 0,C 180,E1 31040.955,E2 31040.955} C_VEL
LIN {X 0,Y 680.851,Z 1141.137,A -85,B 0,C 180,E1 31038.82,E2 31038.82} C_VEL
LIN {X 0,Y 681.364,Z 1126.347,A -85,B 0,C 180,E1 31036.594,E2 31036.594} C_VEL
LIN {X 0,Y 682.005,Z 1110.683,A -85,B 0,C 180,E1 31034.525,E2 31034.525} C_VEL
LIN {X 0,Y 682.866,Z 1092.521,A -85,B 0,C 180,E1 31032.408,E2 31032.408} C_VEL
LIN {X 0,Y 683.791,Z 1073.311,A -85,B 0,C 180,E1 31030.437,E2 31030.437} C_VEL
LIN {X 0,Y 684.966,Z 1052.065,A -85,B 0,C 180,E1 31028.507,E2 31028.507} C_VEL
LIN {X 0,Y 686.221,Z 1029.48,A -85,B 0,C 180,E1 31026.697,E2 31026.697} C_VEL
LIN {X 0,Y 687.588,Z 1006.154,A -85,B 0,C 180,E1 31025.058,E2 31025.058} C_VEL
LIN {X 0,Y 688.957,Z 981.595,A -85,B 0,C 180,E1 31023.542,E2 31023.542} C_VEL
LIN {X 0,Y 690.399,Z 955.64,A -85,B 0,C 180,E1 31022.157,E2 31022.157} C_VEL
LIN {X 0,Y 691.669,Z 931.107,A -85,B 0,C 180,E1 31021.036,E2 31021.036} C_VEL
LIN {X 0,Y 692.712,Z 909.213,A -85,B 0,C 180,E1 31020.171,E2 31020.171} C_VEL
LIN {X 0,Y 693.732,Z 884.766,A -85,B 0,C 180,E1 31019.35,E2 31019.35} C_VEL
LIN {X 0,Y 694.762,Z 856.489,A -85,B 0,C 180,E1 31018.586,E2 31018.586} C_VEL
LIN {X 0,Y 695.486,Z 831.304,A -85,B 0,C 180,E1 31018.068,E2 31018.068} C_VEL
LIN {X 0,Y 696.06,Z 804.14,A -85,B 0,C 180,E1 31017.662,E2 31017.662} C_VEL
LIN {X 0,Y 698.344,Z 583.209,A -85,B 0,C 180,E1 31014.883,E2 31014.883} C_VEL
LIN {X 0,Y 700.72,Z 371.769,A -85,B 0,C 180,E1 31012.138,E2 31012.138} C_VEL
LIN {X 0,Y 700.697,Z 363.446,A -85,B 0,C 180,E1 31012.018,E2 31012.018} C_VEL
LIN {X 0,Y 688.766,Z 345.77,A -85,B 0,C 180,E1 31010.759,E2 31010.759} C_VEL
LIN {X 0,Y 685.367,Z 340.757,A -85,B 0,C 180,E1 31010.382,E2 31010.382} C_VEL
LIN {X 0,Y 681.801,Z 333.016,A -85,B 0,C 180,E1 31009.435,E2 31009.435} C_VEL
LIN {X 0,Y 680.422,Z 329.47,A -85,B 0,C 180,E1 31008.996,E2 31008.996} C_VEL
LIN {X 0,Y 680.43,Z 329.476,A -85,B 0,C 180,E1 31006.547,E2 31006.547} C_VEL
LIN {X 0,Y 680.495,Z 329.463,A -85,B 0,C 180,E1 31003.561,E2 31003.561} C_VEL
LIN {X 0,Y 680.425,Z 329.47,A -85,B 0,C 180,E1 31000.82,E2 31000.82} C_VEL
LIN {X 0,Y 680.427,Z 329.47,A -85,B 0,C 180,E1 30998.433,E2 30998.433} C_VEL
LIN {X 0,Y 680.519,Z 329.464,A -85,B 0,C 180,E1 30995.515,E2 30995.515} C_VEL
LIN {X 0,Y 680.428,Z 329.467,A -85,B 0,C 180,E1 30992.637,E2 30992.637} C_VEL
LIN {X 0,Y 680.431,Z 329.469,A -85,B 0,C 180,E1 30990.17,E2 30990.17} C_VEL
LIN {X 0,Y 680.515,Z 329.443,A -85,B 0,C 180,E1 30987.264,E2 30987.264} C_VEL
LIN {X 0,Y 680.431,Z 329.467,A -85,B 0,C 180,E1 30984.389,E2 30984.389} C_VEL
LIN {X 0,Y 680.432,Z 329.449,A -85,B 0,C 180,E1 30981.916,E2 30981.916} C_VEL
LIN {X 0,Y 680.519,Z 329.465,A -85,B 0,C 180,E1 30979.038,E2 30979.038} C_VEL
LIN {X 0,Y 680.433,Z 329.464,A -85,B 0,C 180,E1 30976.213,E2 30976.213} C_VEL
LIN {X 0,Y 680.434,Z 329.466,A -85,B 0,C 180,E1 30973.761,E2 30973.761} C_VEL
LIN {X 0,Y 680.52,Z 329.461,A -85,B 0,C 180,E1 30970.84,E2 30970.84} C_VEL
LIN {X 0,Y 680.434,Z 329.467,A -85,B 0,C 180,E1 30967.946,E2 30967.946} C_VEL
LIN {X 0,Y 680.44,Z 329.463,A -85,B 0,C 180,E1 30965.481,E2 30965.481} C_VEL
LIN {X 0,Y 680.511,Z 329.46,A -85,B 0,C 180,E1 30962.526,E2 30962.526} C_VEL
LIN {X 0,Y 680.436,Z 329.464,A -85,B 0,C 180,E1 30959.747,E2 30959.747} C_VEL
LIN {X 0,Y 680.44,Z 329.467,A -85,B 0,C 180,E1 30957.305,E2 30957.305} C_VEL
LIN {X 0,Y 680.52,Z 329.465,A -85,B 0,C 180,E1 30954.35,E2 30954.35} C_VEL
LIN {X 0,Y 680.439,Z 329.463,A -85,B 0,C 180,E1 30951.55,E2 30951.55} C_VEL
LIN {X 0,Y 680.44,Z 329.465,A -85,B 0,C 180,E1 30949.073,E2 30949.073} C_VEL
LIN {X 0,Y 680.523,Z 329.444,A -85,B 0,C 180,E1 30946.143,E2 30946.143} C_VEL
LIN {X 0,Y 680.443,Z 329.465,A -85,B 0,C 180,E1 30943.347,E2 30943.347} C_VEL
LIN {X 0,Y 680.446,Z 329.445,A -85,B 0,C 180,E1 30940.782,E2 30940.782} C_VEL
LIN {X 0,Y 680.505,Z 329.462,A -85,B 0,C 180,E1 30937.766,E2 30937.766} C_VEL
LIN {X 0,Y 680.44,Z 329.444,A -85,B 0,C 180,E1 30935.044,E2 30935.044} C_VEL
LIN {X 0,Y 680.454,Z 329.468,A -85,B 0,C 180,E1 30932.522,E2 30932.522} C_VEL
LIN {X 0,Y 680.489,Z 329.461,A -85,B 0,C 180,E1 30929.442,E2 30929.442} C_VEL
LIN {X 0,Y 680.443,Z 329.462,A -85,B 0,C 180,E1 30926.73,E2 30926.73} C_VEL
LIN {X 0,Y 680.486,Z 329.468,A -85,B 0,C 180,E1 30924.002,E2 30924.002} C_VEL
LIN {X 0,Y 680.459,Z 329.474,A -85,B 0,C 180,E1 30920.921,E2 30920.921} C_VEL
LIN {X 0,Y 680.469,Z 329.617,A -85,B 0,C 180,E1 30918.701,E2 30918.701} C_VEL
LIN {X 0,Y 681.568,Z 332.666,A -85,B 0,C 180,E1 30918.35,E2 30918.35} C_VEL
LIN {X 0,Y 682.721,Z 334.809,A -85,B 0,C 180,E1 30918.071,E2 30918.071} C_VEL
LIN {X 0,Y 688.556,Z 347.264,A -85,B 0,C 180,E1 30916.556,E2 30916.556} C_VEL
LIN {X 0,Y 690.59,Z 351.334,A -85,B 0,C 180,E1 30916.104,E2 30916.104} C_VEL
LIN {X 0,Y 698.327,Z 363.134,A -85,B 0,C 180,E1 30915.278,E2 30915.278} C_VEL
LIN {X 0,Y 700.81,Z 373.257,A -85,B 0,C 180,E1 30914.93,E2 30914.93} C_VEL
LIN {X 0,Y 698.421,Z 586.084,A -85,B 0,C 180,E1 30912.163,E2 30912.163} C_VEL
LIN {X 0,Y 696.111,Z 809.17,A -85,B 0,C 180,E1 30909.355,E2 30909.355} C_VEL
LIN {X 0,Y 695.538,Z 840.052,A -85,B 0,C 180,E1 30908.911,E2 30908.911} C_VEL
LIN {X 0,Y 694.783,Z 865.238,A -85,B 0,C 180,E1 30908.397,E2 30908.397} C_VEL
LIN {X 0,Y 693.898,Z 890.9,A -85,B 0,C 180,E1 30907.722,E2 30907.722} C_VEL
LIN {X 0,Y 692.783,Z 917.481,A -85,B 0,C 180,E1 30906.846,E2 30906.846} C_VEL
LIN {X 0,Y 691.789,Z 938.369,A -85,B 0,C 180,E1 30906.032,E2 30906.032} C_VEL
LIN {X 0,Y 690.755,Z 958.667,A -85,B 0,C 180,E1 30905.129,E2 30905.129} C_VEL
LIN {X 0,Y 689.674,Z 978.667,A -85,B 0,C 180,E1 30904.122,E2 30904.122} C_VEL
LIN {X 0,Y 688.522,Z 999.47,A -85,B 0,C 180,E1 30902.945,E2 30902.945} C_VEL
LIN {X 0,Y 687.068,Z 1024.255,A -85,B 0,C 180,E1 30901.349,E2 30901.349} C_VEL
LIN {X 0,Y 685.991,Z 1043.455,A -85,B 0,C 180,E1 30899.947,E2 30899.947} C_VEL
